RoboDK station: kr30 cnc template 7 axis 2.rdk

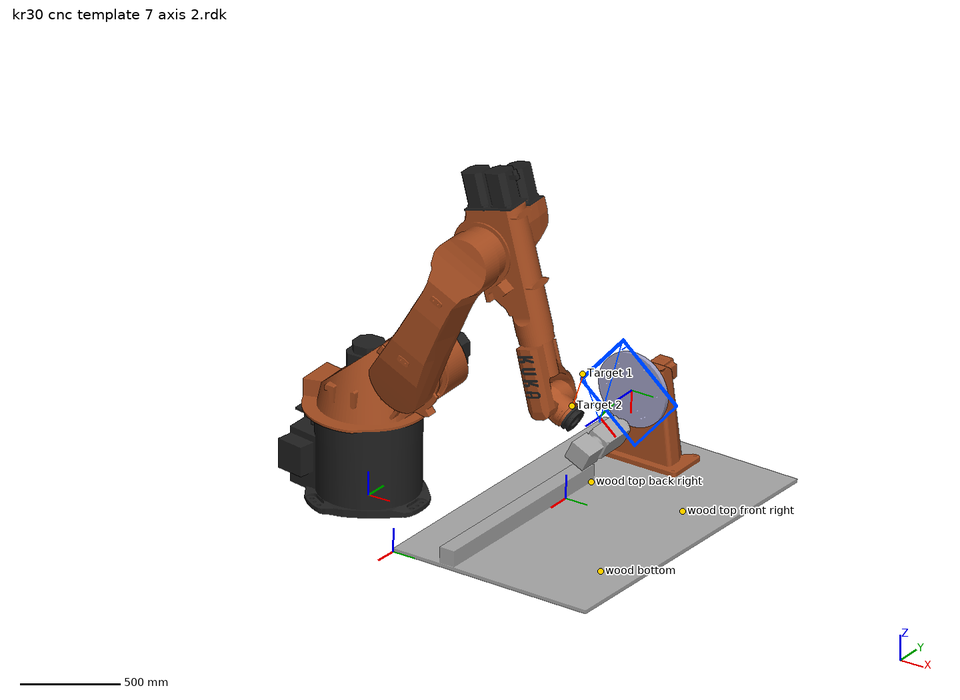
[picture v0: the station drawn from its stored meshes, robots at their saved joint values, targets as dots, program paths as lines]
Station kr30 cnc template 7 axis 2. Poses are relative to the parent item; angles as X-Y-Z fixed-axis rotations.
  - frame KUKA KR 30 HA Base at (0, 0, 0) mm
    - robot KUKA KR 30 HA: 6 axes, payload 30 kg, reach 2033 mm, repeatability 0.05 mm, weight 665 kg
        modified DH rows (alpha deg, a mm, theta deg, d mm): 0, 0, 0, 815; -90, 350, 0, 0; 0, 850, -90, 0; -90, 145, 0, 820; 90, 0, 0, 0; -90, 0, 180, 170
        joint limits [-185, -135, -120, -350, -119, -350] to [185, 35, 158, 350, 119, 350]; home [0, -90, 90, 0, 0, 0]; saved at [-1.685, -62.909, 138.513, -0.146, -48.713, -90.115]
      - tool rc90 spindle mm, TCP at (267.95, 0.68, 160.99) mm, rotated rx 0 ry 90 rz 0 deg, size 110 x 421.3 x 118 mm, geometry from rc90 spindle mm.stl
    - frame Tabletop at (921.82, -1104.91, 385) mm, rotated rx -0.93 ry -0.21 rz -89.9 deg
      - object tabletop CHECK HEIGHT at (-1839.9, 0, 0) mm, size 1839.9 x 1168.4 x 19 mm, geometry from kr30 tabletop mm.stl
      - object kr30 pipe jig base at (-1220, -610.6, 0) mm, size 1217.6 x 88.9 x 88.9 mm, geometry from kr30 pipe jig base.stl
      - frame Frame 3 at (-930, 400, 45) mm
      - target wood top back right (Cartesian target) at (-1141.49, 406.84, 52.26) mm, rotated rx 18.07 ry 89.88 rz 108.17 deg; joints [-2.086, -55.392, 143.759, 178.106, 87.553, -179.775] of KUKA KR 30 HA
      - target wood bottom (Cartesian target) at (-376.62, 995.52, 35.89) mm, rotated rx 18.07 ry 89.88 rz 108.17 deg; joints [24.587, -27.296, 76.752, 211.623, 53.064, -199.759] of KUKA KR 30 HA
      - target wood top front right (Cartesian target) at (-1142.68, 960.22, 52.55) mm, rotated rx 18.06 ry 89.88 rz 108.16 deg; joints [-1.42, -37.516, 98.016, 178.579, 59.693, -179.129] of KUKA KR 30 HA
  - machining project Machining Settings: C:/Users/Research Office/Desktop/paulina a5.apt | rotZ(0) | rotX(0)*rotY(0)
  - frame KUKA KP1 MD250 Base at (1360.87, 339.35, 824.43) mm, rotated rx -93.1 ry 88.62 rz 178.42 deg
    - robot KUKA KP1 MD250: 1 axes, payload 250 kg
        modified DH rows (alpha deg, a mm, theta deg, d mm): 0, 0, 0, 0
        joint limits [-360] to [360]; home [0]; saved at [-57.717]
    - frame Frame 5 at (179.73, -160.64, 39.79) mm, rotated rx 0 ry 0 rz 50 deg
      - target Target 1 (Cartesian target) at (-214.1, 84.73, -7.48) mm, rotated rx -180 ry 0 rz 150.96 deg; joints [-1.66, -91.883, 138.777, -0.061, 23.524, -90.098, -57.717] of KUKA KR 30 HA
      - target Target 2 (Cartesian target) at (-120.32, 1.96, 112.71) mm, rotated rx 180 ry 0 rz 142.66 deg; joints [4.871, -81.16, 137.42, -3.434, 22.572, -80.574, -143.17] of KUKA KR 30 HA
  - program Machining (635 instructions, listed below)
  - program sync move test (5 instructions, listed below)
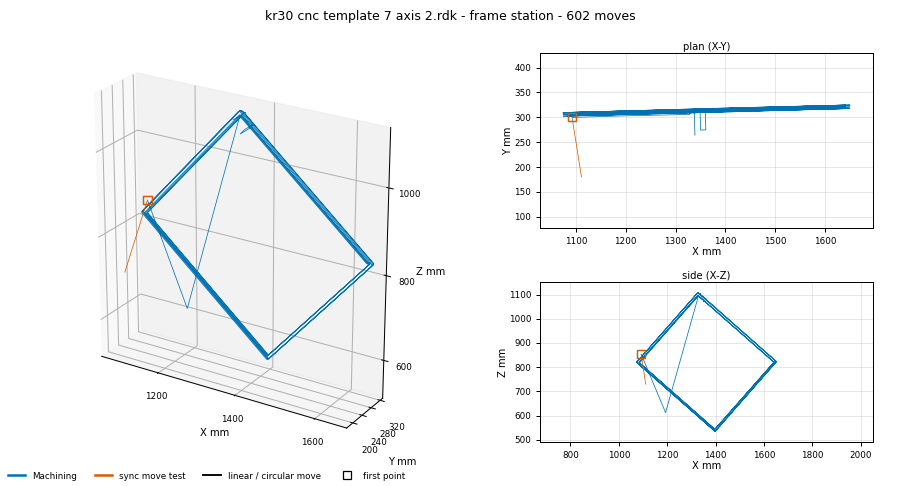
[picture p0: tool path of kr30 cnc template 7 axis 2.rdk in frame station, 602 of 602 moves have a stored position in this frame; points joined in program order, loops and branches not executed]

--- program Machining (robot KUKA KR 30 HA) ---
  Smooth(10)
  Print: /'1001'
  Print: /''
  Print: /'diagonal cut'
  Set speed (100.0 mm/s)
  Set Tool: rc90 spindle mm
  Set Ref.: Frame 5
  Show rc90 spindle mm
  MoveJ 1 to (-214.1, 84.73, -7.48) mm, rotated rx -180 ry 0 rz 150.96 deg; joints [-1.66, -91.883, 138.777, -0.061, 23.524, -90.098, -57.717]
  Set speed (38.1 mm/s)
  MoveL to (21.22, -29.86, -7.48) mm, rotated rx 180 ry 0 rz -151.32 deg; joints [-1.66, -91.883, 138.777, -0.061, 23.524, -90.098, -57.717]
  MoveL 1470 to (-195.61, 421.25, -7.47) mm, rotated rx 180 ry 0 rz 74.1 deg; joints [-1.66, -91.899, 138.812, -0.061, 23.524, -90.098, -57.737]
  Set speed (25.4 mm/s)
  MoveL 1471 to (-195.61, 421.25, -9.84) mm, rotated rx -180 ry 0 rz 74.1 deg; joints [-1.797, -91.898, 138.811, 0.054, 23.524, -90.333, -57.737]
  MoveL 1472 to (-195.61, 421.89, -10.47) mm, rotated rx 180 ry 0 rz 74.1 deg; joints [-1.834, -91.952, 138.836, 0.085, 23.524, -90.397, -57.707]
  Set speed (38.1 mm/s)
  MoveL 1473 to (-194.97, 422.52, -10.48) mm, rotated rx 180 ry 0 rz 74.1 deg; joints [-1.834, -91.991, 138.825, 0.086, 23.524, -90.397, -57.658]
  Set speed (76.2 mm/s)
  MoveL 1474 to (213.41, 422.52, -10.47) mm, rotated rx -180 ry 0 rz 74.1 deg; joints [-1.774, -87.647, 118.581, 0.214, 23.524, -90.444, -41.757]
  MoveL 1475 to (213.89, 422.53, -10.47) mm, rotated rx 180 ry 0 rz 74.1 deg; joints [-1.774, -87.649, 118.56, 0.214, 23.524, -90.445, -41.735]
  MoveL 1476 to (214.13, 422.55, -10.47) mm, rotated rx -180 ry 0 rz 74.1 deg; joints [-1.774, -87.652, 118.551, 0.214, 23.524, -90.445, -41.723]
  MoveL 1477 to (214.37, 422.59, -10.47) mm, rotated rx 180 ry 0 rz 74.1 deg; joints [-1.774, -87.656, 118.543, 0.214, 23.524, -90.445, -41.711]
  MoveL 1478 to (214.61, 422.65, -10.47) mm, rotated rx -180 ry 0 rz 74.1 deg; joints [-1.774, -87.662, 118.536, 0.215, 23.524, -90.445, -41.698]
  MoveL 1479 to (214.85, 422.74, -10.47) mm, rotated rx -180 ry 0 rz 74.1 deg; joints [-1.774, -87.67, 118.531, 0.215, 23.524, -90.445, -41.684]
  MoveL 1480 to (215.09, 422.84, -10.47) mm, rotated rx 180 ry 0 rz 74.1 deg; joints [-1.774, -87.68, 118.526, 0.215, 23.524, -90.445, -41.67]
  MoveL 1481 to (215.34, 422.97, -10.47) mm, rotated rx -180 ry 0 rz 74.1 deg; joints [-1.774, -87.691, 118.522, 0.215, 23.524, -90.445, -41.654]
  MoveL 1482 to (215.58, 423.13, -10.48) mm, rotated rx -180 ry 0 rz 74.1 deg; joints [-1.774, -87.706, 118.521, 0.215, 23.524, -90.445, -41.638]
  MoveL 1483 to (215.82, 423.33, -10.47) mm, rotated rx -180 ry 0 rz 74.1 deg; joints [-1.774, -87.723, 118.521, 0.215, 23.524, -90.446, -41.621]
  MoveL 1484 to (215.96, 423.46, -10.48) mm, rotated rx 180 ry 0 rz 74.1 deg; joints [-1.774, -87.735, 118.521, 0.216, 23.525, -90.446, -41.611]
  MoveL 1485 to (216.09, 423.6, -10.48) mm, rotated rx -180 ry 0 rz 74.1 deg; joints [-1.774, -87.745, 118.521, 0.216, 23.528, -90.446, -41.603]
  MoveL 1486 to (216.2, 423.73, -10.48) mm, rotated rx -180 ry 0 rz 74.1 deg; joints [-1.774, -87.756, 118.521, 0.216, 23.532, -90.446, -41.596]
  MoveL 1487 to (216.3, 423.87, -10.48) mm, rotated rx -180 ry 0 rz 74.1 deg; joints [-1.774, -87.766, 118.521, 0.216, 23.536, -90.446, -41.59]
  MoveL 1488 to (216.39, 424.01, -10.47) mm, rotated rx -180 ry 0 rz 74.1 deg; joints [-1.774, -87.776, 118.521, 0.216, 23.541, -90.446, -41.586]
  MoveL 1489 to (216.47, 424.15, -10.47) mm, rotated rx -180 ry 0 rz 74.1 deg; joints [-1.774, -87.786, 118.521, 0.216, 23.547, -90.446, -41.582]
  MoveL 1490 to (216.69, 424.27, -10.47) mm, rotated rx 180 ry 0 rz 74.1 deg; joints [-1.774, -87.797, 118.518, 0.216, 23.547, -90.446, -41.568]
  MoveL 1491 to (219.83, 424.27, -10.48) mm, rotated rx -180 ry 0 rz 74.1 deg; joints [-1.774, -87.806, 118.385, 0.217, 23.547, -90.447, -41.425]
  MoveL 1492 to (220.05, 424.15, -10.47) mm, rotated rx -180 ry 0 rz 74.1 deg; joints [-1.774, -87.797, 118.369, 0.217, 23.547, -90.447, -41.419]
  MoveL 1493 to (220.05, 53.41, -10.48) mm, rotated rx 180 ry 0 rz 74.1 deg; joints [-1.728, -59.035, 99.349, 0.059, 23.547, -90.273, -51.16]
  MoveL 1494 to (219.83, 53.18, -10.47) mm, rotated rx 180 ry 0 rz 74.1 deg; joints [-1.728, -59.018, 99.35, 0.059, 23.547, -90.272, -51.179]
  MoveL 1495 to (-199.12, 53.18, -10.48) mm, rotated rx 180 ry 0 rz 74.1 deg; joints [-1.791, -64.086, 127.611, -0.153, 23.547, -90.132, -74.372]
  MoveL 1496 to (-199.7, 53.17, -10.48) mm, rotated rx -180 ry 0 rz 74.1 deg; joints [-1.791, -64.101, 127.652, -0.153, 23.547, -90.132, -74.398]
  MoveL 1497 to (-199.9, 53.41, -10.48) mm, rotated rx -180 ry 0 rz 74.1 deg; joints [-1.791, -64.122, 127.672, -0.153, 23.545, -90.132, -74.394]
  MoveL 1498 to (-199.9, 424.15, -10.48) mm, rotated rx -180 ry 0 rz 74.1 deg; joints [-1.835, -92.249, 139.152, 0.086, 23.545, -90.399, -57.747]
  MoveL 1499 to (-199.7, 424.27, -10.48) mm, rotated rx 180 ry 0 rz 74.1 deg; joints [-1.835, -92.255, 139.146, 0.086, 23.545, -90.399, -57.735]
  MoveL 1500 to (-198.11, 424.27, -10.48) mm, rotated rx -180 ry 0 rz 74.1 deg; joints [-1.835, -92.216, 139.057, 0.086, 23.545, -90.399, -57.686]
  MoveL 1501 to (-197.87, 424.15, -10.47) mm, rotated rx -180 ry 0 rz 74.1 deg; joints [-1.835, -92.2, 139.04, 0.086, 23.545, -90.399, -57.685]
  MoveL 1502 to (-197.73, 423.93, -10.48) mm, rotated rx 180 ry 0 rz 74.1 deg; joints [-1.835, -92.178, 139.024, 0.086, 23.545, -90.399, -57.691]
  MoveL 1503 to (-197.57, 423.71, -10.48) mm, rotated rx -180 ry 0 rz 74.1 deg; joints [-1.835, -92.155, 139.006, 0.086, 23.545, -90.398, -57.696]
  MoveL 1504 to (-197.38, 423.49, -10.48) mm, rotated rx 180 ry 0 rz 74.1 deg; joints [-1.835, -92.131, 138.987, 0.086, 23.545, -90.398, -57.7]
  MoveL 1505 to (-197.14, 423.27, -10.47) mm, rotated rx -180 ry 0 rz 74.1 deg; joints [-1.834, -92.107, 138.966, 0.086, 23.545, -90.398, -57.703]
  MoveL 1506 to (-196.96, 423.13, -10.48) mm, rotated rx 180 ry 0 rz 74.1 deg; joints [-1.834, -92.09, 138.95, 0.086, 23.545, -90.398, -57.704]
  MoveL 1507 to (-196.78, 423, -10.47) mm, rotated rx -180 ry 0 rz 74.1 deg; joints [-1.834, -92.076, 138.935, 0.086, 23.545, -90.398, -57.704]
  MoveL 1508 to (-196.6, 422.9, -10.48) mm, rotated rx -180 ry 0 rz 74.1 deg; joints [-1.834, -92.062, 138.921, 0.086, 23.545, -90.398, -57.704]
  MoveL 1509 to (-196.42, 422.81, -10.48) mm, rotated rx -180 ry 0 rz 74.1 deg; joints [-1.834, -92.05, 138.908, 0.086, 23.545, -90.397, -57.702]
  MoveL 1510 to (-196.18, 422.71, -10.47) mm, rotated rx 180 ry 0 rz 74.1 deg; joints [-1.834, -92.036, 138.891, 0.086, 23.545, -90.397, -57.699]
  MoveL 1511 to (-195.93, 422.63, -10.48) mm, rotated rx 180 ry 0 rz 74.1 deg; joints [-1.834, -92.023, 138.874, 0.086, 23.545, -90.397, -57.696]
  MoveL 1512 to (-195.69, 422.58, -10.48) mm, rotated rx 180 ry 0 rz 74.1 deg; joints [-1.834, -92.013, 138.859, 0.086, 23.545, -90.397, -57.691]
  MoveL 1513 to (-195.45, 422.54, -10.48) mm, rotated rx 180 ry 0 rz 74.1 deg; joints [-1.834, -92.004, 138.844, 0.086, 23.545, -90.397, -57.685]
  MoveL 1514 to (-195.21, 422.52, -10.48) mm, rotated rx 180 ry 0 rz 74.1 deg; joints [-1.834, -91.996, 138.83, 0.086, 23.545, -90.397, -57.678]
  MoveL 1515 to (-194.97, 422.52, -10.48) mm, rotated rx -180 ry 0 rz 74.1 deg; joints [-1.834, -91.99, 138.817, 0.086, 23.545, -90.397, -57.671]
  Set speed (38.1 mm/s)
  MoveL 1516 to (-194.97, 421.25, -10.47) mm, rotated rx -180 ry 0 rz 74.1 deg; joints [-1.833, -91.882, 138.768, 0.085, 23.545, -90.396, -57.73]
  MoveL 1517 to (-195.61, 421.25, -10.48) mm, rotated rx -180 ry 0 rz 74.1 deg; joints [-1.834, -91.897, 138.803, 0.084, 23.545, -90.396, -57.75]
  Set speed (25.4 mm/s)
  MoveL 1518 to (-195.61, 421.25, -12.84) mm, rotated rx -180 ry 0 rz 74.1 deg; joints [-1.971, -91.896, 138.802, 0.199, 23.545, -90.631, -57.75]
  MoveL 1519 to (-195.61, 421.89, -13.47) mm, rotated rx -180 ry 0 rz 74.1 deg; joints [-2.008, -91.95, 138.826, 0.231, 23.545, -90.694, -57.72]
  Set speed (38.1 mm/s)
  MoveL 1520 to (-194.97, 422.52, -13.47) mm, rotated rx -180 ry 0 rz 74.1 deg; joints [-2.008, -91.989, 138.815, 0.232, 23.545, -90.695, -57.671]
  Set speed (76.2 mm/s)
  MoveL 1521 to (213.41, 422.52, -13.47) mm, rotated rx -180 ry 0 rz 74.1 deg; joints [-1.922, -87.638, 118.566, 0.429, 23.545, -90.761, -41.772]
  MoveL 1522 to (213.89, 422.53, -13.47) mm, rotated rx -180 ry 0 rz 74.1 deg; joints [-1.921, -87.64, 118.546, 0.429, 23.545, -90.762, -41.75]
  MoveL 1523 to (214.13, 422.55, -13.47) mm, rotated rx 180 ry 0 rz 74.1 deg; joints [-1.921, -87.642, 118.537, 0.429, 23.545, -90.762, -41.738]
  MoveL 1524 to (214.37, 422.59, -13.47) mm, rotated rx 180 ry 0 rz 74.1 deg; joints [-1.921, -87.647, 118.529, 0.429, 23.545, -90.762, -41.726]
  MoveL 1525 to (214.61, 422.65, -13.47) mm, rotated rx -180 ry 0 rz 74.1 deg; joints [-1.921, -87.653, 118.522, 0.429, 23.545, -90.762, -41.713]
  MoveL 1526 to (214.85, 422.74, -13.47) mm, rotated rx 180 ry 0 rz 74.1 deg; joints [-1.921, -87.66, 118.516, 0.43, 23.545, -90.762, -41.7]
  MoveL 1527 to (215.09, 422.84, -13.47) mm, rotated rx 180 ry 0 rz 74.1 deg; joints [-1.921, -87.67, 118.511, 0.43, 23.545, -90.762, -41.685]
  MoveL 1528 to (215.34, 422.97, -13.48) mm, rotated rx -180 ry 0 rz 74.1 deg; joints [-1.921, -87.682, 118.508, 0.43, 23.545, -90.763, -41.67]
  MoveL 1529 to (215.58, 423.13, -13.47) mm, rotated rx 180 ry 0 rz 74.1 deg; joints [-1.921, -87.696, 118.506, 0.43, 23.545, -90.763, -41.654]
  MoveL 1530 to (215.82, 423.33, -13.47) mm, rotated rx -180 ry 0 rz 74.1 deg; joints [-1.922, -87.714, 118.506, 0.431, 23.545, -90.763, -41.636]
  MoveL 1531 to (215.96, 423.46, -13.47) mm, rotated rx -180 ry 0 rz 74.1 deg; joints [-1.922, -87.725, 118.506, 0.431, 23.547, -90.763, -41.626]
  MoveL 1532 to (216.09, 423.6, -13.47) mm, rotated rx -180 ry 0 rz 74.1 deg; joints [-1.922, -87.736, 118.506, 0.431, 23.549, -90.763, -41.618]
  MoveL 1533 to (216.2, 423.73, -13.47) mm, rotated rx 180 ry 0 rz 74.1 deg; joints [-1.922, -87.747, 118.507, 0.431, 23.552, -90.763, -41.611]
  MoveL 1534 to (216.3, 423.87, -13.47) mm, rotated rx -180 ry 0 rz 74.1 deg; joints [-1.922, -87.757, 118.507, 0.431, 23.557, -90.763, -41.605]
  MoveL 1535 to (216.39, 424.01, -13.47) mm, rotated rx -180 ry 0 rz 74.1 deg; joints [-1.922, -87.767, 118.507, 0.431, 23.562, -90.763, -41.601]
  MoveL 1536 to (216.47, 424.15, -13.47) mm, rotated rx -180 ry 0 rz 74.1 deg; joints [-1.922, -87.776, 118.507, 0.431, 23.568, -90.763, -41.597]
  MoveL 1537 to (216.69, 424.27, -13.47) mm, rotated rx -180 ry 0 rz 74.1 deg; joints [-1.922, -87.787, 118.504, 0.432, 23.568, -90.764, -41.583]
  MoveL 1538 to (219.83, 424.27, -13.47) mm, rotated rx -180 ry 0 rz 74.1 deg; joints [-1.921, -87.797, 118.371, 0.433, 23.568, -90.765, -41.441]
  MoveL 1539 to (220.05, 424.15, -13.47) mm, rotated rx -180 ry 0 rz 74.1 deg; joints [-1.921, -87.788, 118.355, 0.433, 23.567, -90.765, -41.434]
  MoveL 1540 to (220.05, 53.41, -13.48) mm, rotated rx -180 ry 0 rz 74.1 deg; joints [-1.843, -59.027, 99.34, 0.185, 23.567, -90.49, -51.179]
  MoveL 1541 to (219.83, 53.18, -13.47) mm, rotated rx -180 ry 0 rz 74.1 deg; joints [-1.843, -59.01, 99.341, 0.185, 23.567, -90.49, -51.198]
  MoveL 1542 to (-197.29, 53.18, -13.48) mm, rotated rx -180 ry 0 rz 74.1 deg; joints [-1.931, -64.037, 127.476, -0.133, 23.567, -90.29, -74.307]
  MoveL 1543 to (-197.94, 53.18, -13.48) mm, rotated rx 180 ry 0 rz 74.1 deg; joints [-1.932, -64.054, 127.523, -0.134, 23.567, -90.29, -74.336]
  MoveL 1544 to (-198.16, 53.41, -13.48) mm, rotated rx -180 ry 0 rz 74.1 deg; joints [-1.932, -64.076, 127.544, -0.134, 23.567, -90.29, -74.335]
  MoveL 1545 to (-198.16, 424.15, -13.48) mm, rotated rx -180 ry 0 rz 74.1 deg; joints [-2.01, -92.205, 139.045, 0.232, 23.567, -90.697, -57.707]
  MoveL 1546 to (-198.01, 424.27, -13.48) mm, rotated rx -180 ry 0 rz 74.1 deg; joints [-2.01, -92.211, 139.042, 0.233, 23.567, -90.698, -57.697]
  MoveL 1547 to (-197.87, 424.15, -13.47) mm, rotated rx -180 ry 0 rz 74.1 deg; joints [-2.009, -92.198, 139.029, 0.233, 23.567, -90.697, -57.698]
  MoveL 1548 to (-197.73, 423.93, -13.47) mm, rotated rx -180 ry 0 rz 74.1 deg; joints [-2.009, -92.176, 139.013, 0.232, 23.567, -90.697, -57.705]
  MoveL 1549 to (-197.57, 423.71, -13.48) mm, rotated rx -180 ry 0 rz 74.1 deg; joints [-2.009, -92.153, 138.996, 0.232, 23.567, -90.697, -57.71]
  MoveL 1550 to (-197.38, 423.49, -13.48) mm, rotated rx -180 ry 0 rz 74.1 deg; joints [-2.009, -92.129, 138.977, 0.232, 23.567, -90.696, -57.714]
  MoveL 1551 to (-197.22, 423.33, -13.47) mm, rotated rx 180 ry 0 rz 74.1 deg; joints [-2.009, -92.112, 138.962, 0.232, 23.567, -90.696, -57.716]
  MoveL 1552 to (-197.14, 423.27, -13.48) mm, rotated rx -180 ry 0 rz 74.1 deg; joints [-2.009, -92.105, 138.955, 0.232, 23.567, -90.696, -57.717]
  MoveL 1553 to (-196.96, 423.13, -13.48) mm, rotated rx -180 ry 0 rz 74.1 deg; joints [-2.009, -92.088, 138.94, 0.232, 23.567, -90.696, -57.718]
  MoveL 1554 to (-196.78, 423, -13.47) mm, rotated rx -180 ry 0 rz 74.1 deg; joints [-2.009, -92.073, 138.925, 0.231, 23.567, -90.696, -57.718]
  MoveL 1555 to (-196.6, 422.9, -13.47) mm, rotated rx -180 ry 0 rz 74.1 deg; joints [-2.008, -92.06, 138.911, 0.231, 23.567, -90.695, -57.718]
  MoveL 1556 to (-196.42, 422.81, -13.47) mm, rotated rx 180 ry 0 rz 74.1 deg; joints [-2.008, -92.048, 138.897, 0.231, 23.567, -90.695, -57.716]
  MoveL 1557 to (-196.18, 422.71, -13.47) mm, rotated rx -180 ry 0 rz 74.1 deg; joints [-2.008, -92.034, 138.88, 0.231, 23.567, -90.695, -57.713]
  MoveL 1558 to (-195.93, 422.63, -13.47) mm, rotated rx 180 ry 0 rz 74.1 deg; joints [-2.008, -92.021, 138.864, 0.231, 23.567, -90.695, -57.709]
  MoveL 1559 to (-195.69, 422.58, -13.47) mm, rotated rx -180 ry 0 rz 74.1 deg; joints [-2.008, -92.011, 138.849, 0.231, 23.567, -90.695, -57.705]
  MoveL 1560 to (-195.45, 422.54, -13.48) mm, rotated rx 180 ry 0 rz 74.1 deg; joints [-2.008, -92.002, 138.834, 0.231, 23.567, -90.695, -57.699]
  MoveL 1561 to (-195.21, 422.52, -13.48) mm, rotated rx -180 ry 0 rz 74.1 deg; joints [-2.008, -91.994, 138.82, 0.231, 23.567, -90.695, -57.692]
  MoveL 1562 to (-194.97, 422.52, -13.47) mm, rotated rx 180 ry 0 rz 74.1 deg; joints [-2.008, -91.988, 138.806, 0.232, 23.567, -90.695, -57.685]
  Set speed (38.1 mm/s)
  MoveL 1563 to (-194.97, 421.25, -13.47) mm, rotated rx -180 ry 0 rz 74.1 deg; joints [-2.007, -91.88, 138.757, 0.23, 23.567, -90.693, -57.744]
  MoveL 1564 to (-195.61, 421.25, -13.47) mm, rotated rx 180 ry 0 rz 74.1 deg; joints [-2.008, -91.895, 138.792, 0.23, 23.567, -90.693, -57.764]
  Set speed (25.4 mm/s)
  MoveL 1565 to (-195.61, 421.25, -15.84) mm, rotated rx 180 ry 0 rz 74.1 deg; joints [-2.145, -91.894, 138.791, 0.344, 23.567, -90.927, -57.764]
  MoveL 1566 to (-195.61, 421.89, -16.48) mm, rotated rx 180 ry 0 rz 74.1 deg; joints [-2.182, -91.948, 138.815, 0.376, 23.567, -90.992, -57.734]
  Set speed (38.1 mm/s)
  MoveL 1567 to (-194.97, 422.52, -16.47) mm, rotated rx 180 ry 0 rz 74.1 deg; joints [-2.182, -91.986, 138.805, 0.378, 23.567, -90.993, -57.684]
  Set speed (76.2 mm/s)
  MoveL 1568 to (213.41, 422.52, -16.47) mm, rotated rx -180 ry 0 rz 74.1 deg; joints [-2.069, -87.627, 118.551, 0.643, 23.567, -91.078, -41.789]
  MoveL 1569 to (213.89, 422.53, -16.47) mm, rotated rx -180 ry 0 rz 74.1 deg; joints [-2.069, -87.629, 118.531, 0.643, 23.568, -91.078, -41.767]
  MoveL 1570 to (214.13, 422.55, -16.47) mm, rotated rx -180 ry 0 rz 74.1 deg; joints [-2.069, -87.632, 118.522, 0.643, 23.567, -91.078, -41.755]
  MoveL 1571 to (214.37, 422.59, -16.47) mm, rotated rx -180 ry 0 rz 74.1 deg; joints [-2.069, -87.636, 118.514, 0.643, 23.567, -91.078, -41.743]
  MoveL 1572 to (214.61, 422.65, -16.47) mm, rotated rx 180 ry 0 rz 74.1 deg; joints [-2.069, -87.642, 118.507, 0.644, 23.567, -91.078, -41.73]
  MoveL 1573 to (214.85, 422.74, -16.47) mm, rotated rx 180 ry 0 rz 74.1 deg; joints [-2.069, -87.65, 118.501, 0.644, 23.567, -91.079, -41.716]
  MoveL 1574 to (215.09, 422.84, -16.48) mm, rotated rx 180 ry 0 rz 74.1 deg; joints [-2.069, -87.66, 118.496, 0.644, 23.567, -91.079, -41.701]
  MoveL 1575 to (215.34, 422.97, -16.47) mm, rotated rx -180 ry 0 rz 74.1 deg; joints [-2.069, -87.672, 118.493, 0.645, 23.567, -91.079, -41.686]
  MoveL 1576 to (215.58, 423.13, -16.47) mm, rotated rx -180 ry 0 rz 74.1 deg; joints [-2.069, -87.686, 118.491, 0.645, 23.567, -91.08, -41.67]
  MoveL 1577 to (215.82, 423.33, -16.47) mm, rotated rx -180 ry 0 rz 74.1 deg; joints [-2.069, -87.703, 118.491, 0.646, 23.567, -91.08, -41.652]
  MoveL 1578 to (215.96, 423.46, -16.47) mm, rotated rx 180 ry 0 rz 74.1 deg; joints [-2.069, -87.715, 118.491, 0.646, 23.569, -91.08, -41.643]
  MoveL 1579 to (216.09, 423.6, -16.48) mm, rotated rx 180 ry 0 rz 74.1 deg; joints [-2.069, -87.726, 118.491, 0.646, 23.572, -91.08, -41.634]
  MoveL 1580 to (216.2, 423.73, -16.47) mm, rotated rx -180 ry 0 rz 74.1 deg; joints [-2.069, -87.736, 118.491, 0.646, 23.575, -91.08, -41.627]
  MoveL 1581 to (216.3, 423.87, -16.47) mm, rotated rx -180 ry 0 rz 74.1 deg; joints [-2.069, -87.746, 118.491, 0.646, 23.579, -91.08, -41.622]
  MoveL 1582 to (216.39, 424.01, -16.47) mm, rotated rx -180 ry 0 rz 74.1 deg; joints [-2.07, -87.756, 118.491, 0.646, 23.584, -91.08, -41.617]
  MoveL 1583 to (216.47, 424.15, -16.48) mm, rotated rx 180 ry 0 rz 74.1 deg; joints [-2.07, -87.766, 118.491, 0.646, 23.59, -91.08, -41.613]
  MoveL 1584 to (216.69, 424.27, -16.47) mm, rotated rx 180 ry 0 rz 74.1 deg; joints [-2.07, -87.777, 118.488, 0.646, 23.59, -91.081, -41.599]
  MoveL 1585 to (219.83, 424.27, -16.47) mm, rotated rx -180 ry 0 rz 74.1 deg; joints [-2.069, -87.787, 118.356, 0.649, 23.59, -91.082, -41.457]
  MoveL 1586 to (220.05, 424.15, -16.47) mm, rotated rx 180 ry 0 rz 74.1 deg; joints [-2.069, -87.777, 118.34, 0.649, 23.589, -91.082, -41.45]
  MoveL 1587 to (220.05, 53.41, -16.48) mm, rotated rx 180 ry 0 rz 74.1 deg; joints [-1.957, -59.019, 99.329, 0.31, 23.589, -90.707, -51.199]
  MoveL 1588 to (219.83, 53.17, -16.48) mm, rotated rx -180 ry 0 rz 74.1 deg; joints [-1.957, -59.001, 99.33, 0.309, 23.589, -90.707, -51.218]
  MoveL 1589 to (-196.42, 53.18, -16.48) mm, rotated rx 180 ry 0 rz 74.1 deg; joints [-2.072, -64.014, 127.409, -0.114, 23.589, -90.448, -74.285]
  MoveL 1590 to (-196.42, 53.41, -16.48) mm, rotated rx 180 ry 0 rz 74.1 deg; joints [-2.072, -64.03, 127.415, -0.114, 23.589, -90.448, -74.275]
  MoveL 1591 to (-196.42, 422.66, -16.48) mm, rotated rx -180 ry 0 rz 74.1 deg; joints [-2.183, -92.032, 138.881, 0.376, 23.589, -90.992, -57.737]
  MoveL 1592 to (-196.42, 422.81, -16.48) mm, rotated rx 180 ry 0 rz 74.1 deg; joints [-2.183, -92.045, 138.887, 0.377, 23.589, -90.993, -57.73]
  MoveL 1593 to (-196.18, 422.71, -16.48) mm, rotated rx 180 ry 0 rz 74.1 deg; joints [-2.182, -92.031, 138.87, 0.377, 23.589, -90.992, -57.727]
  MoveL 1594 to (-195.93, 422.63, -16.48) mm, rotated rx -180 ry 0 rz 74.1 deg; joints [-2.182, -92.018, 138.853, 0.377, 23.589, -90.992, -57.723]
  MoveL 1595 to (-195.69, 422.58, -16.47) mm, rotated rx -180 ry 0 rz 74.1 deg; joints [-2.182, -92.008, 138.838, 0.377, 23.589, -90.992, -57.718]
  MoveL 1596 to (-195.45, 422.54, -16.48) mm, rotated rx 180 ry 0 rz 74.1 deg; joints [-2.182, -91.999, 138.823, 0.377, 23.589, -90.992, -57.712]
  MoveL 1597 to (-195.21, 422.52, -16.48) mm, rotated rx -180 ry 0 rz 74.1 deg; joints [-2.182, -91.992, 138.809, 0.377, 23.589, -90.992, -57.706]
  MoveL 1598 to (-194.97, 422.52, -16.47) mm, rotated rx 180 ry 0 rz 74.1 deg; joints [-2.182, -91.986, 138.796, 0.377, 23.589, -90.992, -57.698]
  MoveL 1599 to (-164.9, 422.52, -17.53) mm, rotated rx 180 ry 0 rz 74.1 deg; joints [-2.229, -91.287, 137.144, 0.445, 23.589, -91.095, -56.745]
  MoveL 1600 to (213.41, 422.52, -17.52) mm, rotated rx -180 ry 0 rz 74.1 deg; joints [-2.121, -87.618, 118.537, 0.717, 23.589, -91.188, -41.805]
  MoveL 1601 to (213.89, 422.53, -17.52) mm, rotated rx 180 ry 0 rz 74.1 deg; joints [-2.121, -87.62, 118.516, 0.717, 23.589, -91.188, -41.783]
  MoveL 1602 to (214.13, 422.55, -17.52) mm, rotated rx -180 ry 0 rz 74.1 deg; joints [-2.121, -87.622, 118.507, 0.717, 23.589, -91.188, -41.771]
  MoveL 1603 to (214.37, 422.59, -17.52) mm, rotated rx -180 ry 0 rz 74.1 deg; joints [-2.121, -87.627, 118.499, 0.717, 23.589, -91.188, -41.759]
  MoveL 1604 to (214.61, 422.65, -17.52) mm, rotated rx 180 ry 0 rz 74.1 deg; joints [-2.121, -87.633, 118.492, 0.718, 23.589, -91.188, -41.746]
  MoveL 1605 to (214.85, 422.74, -17.52) mm, rotated rx -180 ry 0 rz 74.1 deg; joints [-2.121, -87.641, 118.486, 0.718, 23.589, -91.189, -41.732]
  MoveL 1606 to (215.09, 422.84, -17.52) mm, rotated rx 180 ry 0 rz 74.1 deg; joints [-2.121, -87.65, 118.482, 0.718, 23.589, -91.189, -41.718]
  MoveL 1607 to (215.34, 422.97, -17.52) mm, rotated rx -180 ry 0 rz 74.1 deg; joints [-2.121, -87.662, 118.478, 0.719, 23.589, -91.189, -41.703]
  MoveL 1608 to (215.58, 423.13, -17.52) mm, rotated rx -180 ry 0 rz 74.1 deg; joints [-2.121, -87.676, 118.476, 0.719, 23.589, -91.19, -41.686]
  MoveL 1609 to (215.82, 423.33, -17.52) mm, rotated rx -180 ry 0 rz 74.1 deg; joints [-2.121, -87.694, 118.476, 0.72, 23.589, -91.19, -41.669]
  MoveL 1610 to (215.96, 423.46, -17.52) mm, rotated rx -180 ry 0 rz 74.1 deg; joints [-2.121, -87.705, 118.476, 0.72, 23.591, -91.19, -41.659]
  MoveL 1611 to (216.09, 423.6, -17.52) mm, rotated rx 180 ry 0 rz 74.1 deg; joints [-2.121, -87.716, 118.476, 0.72, 23.594, -91.19, -41.651]
  MoveL 1612 to (216.2, 423.73, -17.52) mm, rotated rx 180 ry 0 rz 74.1 deg; joints [-2.121, -87.727, 118.477, 0.72, 23.597, -91.19, -41.644]
  MoveL 1613 to (216.3, 423.87, -17.52) mm, rotated rx 180 ry 0 rz 74.1 deg; joints [-2.121, -87.737, 118.477, 0.72, 23.601, -91.191, -41.638]
  MoveL 1614 to (216.39, 424.01, -17.52) mm, rotated rx -180 ry 0 rz 74.1 deg; joints [-2.121, -87.747, 118.477, 0.72, 23.606, -91.191, -41.633]
  MoveL 1615 to (216.47, 424.15, -17.52) mm, rotated rx -180 ry 0 rz 74.1 deg; joints [-2.121, -87.756, 118.477, 0.72, 23.612, -91.191, -41.629]
  MoveL 1616 to (216.69, 424.27, -17.52) mm, rotated rx 180 ry 0 rz 74.1 deg; joints [-2.121, -87.767, 118.474, 0.721, 23.612, -91.191, -41.615]
  MoveL 1617 to (219.83, 424.27, -17.52) mm, rotated rx 180 ry 0 rz 74.1 deg; joints [-2.121, -87.777, 118.341, 0.723, 23.612, -91.192, -41.473]
  MoveL 1618 to (220.05, 424.15, -17.52) mm, rotated rx 180 ry 0 rz 74.1 deg; joints [-2.121, -87.768, 118.326, 0.724, 23.612, -91.192, -41.466]
  MoveL 1619 to (220.05, 53.41, -17.52) mm, rotated rx -180 ry 0 rz 74.1 deg; joints [-1.996, -59.01, 99.319, 0.353, 23.612, -90.782, -51.22]
  MoveL 1620 to (219.83, 53.18, -17.52) mm, rotated rx 180 ry 0 rz 74.1 deg; joints [-1.996, -58.993, 99.321, 0.352, 23.612, -90.782, -51.239]
  MoveL 1621 to (-195.15, 53.18, -17.53) mm, rotated rx 180 ry 0 rz 74.1 deg; joints [-2.121, -63.98, 127.315, -0.107, 23.612, -90.504, -74.247]
  MoveL 1622 to (-195.65, 53.17, -17.52) mm, rotated rx 180 ry 0 rz 74.1 deg; joints [-2.121, -63.994, 127.351, -0.107, 23.612, -90.504, -74.269]
  MoveL 1623 to (-195.81, 53.41, -17.52) mm, rotated rx -180 ry 0 rz 74.1 deg; joints [-2.121, -64.014, 127.368, -0.107, 23.612, -90.504, -74.266]
  MoveL 1624 to (-195.81, 422.38, -17.53) mm, rotated rx -180 ry 0 rz 74.1 deg; joints [-2.243, -91.992, 138.827, 0.426, 23.612, -91.095, -57.745]
  MoveL 1625 to (-195.65, 422.57, -17.52) mm, rotated rx -180 ry 0 rz 74.1 deg; joints [-2.243, -92.004, 138.825, 0.427, 23.612, -91.095, -57.731]
  MoveL 1626 to (-195.48, 422.55, -17.52) mm, rotated rx -180 ry 0 rz 74.1 deg; joints [-2.243, -91.998, 138.815, 0.427, 23.612, -91.095, -57.727]
  MoveL 1627 to (-195.32, 422.53, -17.52) mm, rotated rx -180 ry 0 rz 74.1 deg; joints [-2.243, -91.993, 138.805, 0.427, 23.612, -91.095, -57.723]
  MoveL 1628 to (-195.15, 422.52, -17.53) mm, rotated rx 180 ry 0 rz 74.1 deg; joints [-2.243, -91.988, 138.796, 0.427, 23.612, -91.095, -57.718]
  MoveL 1629 to (-194.97, 422.52, -17.53) mm, rotated rx -180 ry 0 rz 74.1 deg; joints [-2.243, -91.984, 138.786, 0.427, 23.612, -91.095, -57.713]
  MoveL 1630 to (-164.9, 422.52, -17.52) mm, rotated rx 180 ry 0 rz 74.1 deg; joints [-2.229, -91.286, 137.134, 0.444, 23.612, -91.094, -56.759]
  Set speed (38.1 mm/s)
  MoveL 1631 to (-164.28, 421.77, -17.52) mm, rotated rx -180 ry 0 rz 74.1 deg; joints [-2.228, -91.208, 137.071, 0.443, 23.612, -91.093, -56.774]
  MoveL 1632 to (-164.81, 418.84, -17.52) mm, rotated rx 180 ry 0 rz 74.1 deg; joints [-2.226, -90.969, 136.984, 0.437, 23.612, -91.087, -56.926]
  MoveL 1633 to (-164.93, 418.21, -16.89) mm, rotated rx 180 ry 0 rz 74.1 deg; joints [-2.19, -90.919, 136.966, 0.405, 23.612, -91.023, -56.958]
  Set speed (100.0 mm/s)
  MoveL 1634 to (-164.93, 418.21, 24.52) mm, rotated rx -180 ry 0 rz 74.1 deg; joints [0.159, -90.892, 136.949, -1.635, 23.612, -86.951, -56.95]
  MoveL 1635 to (-164.87, 434.05, 24.53) mm, rotated rx -180 ry 0 rz 74.1 deg; joints [0.183, -92.247, 137.575, -1.706, 23.612, -86.872, -56.219]
  MoveL 1636 to (-164.87, 434.05, -6.52) mm, rotated rx -180 ry 0 rz 74.1 deg; joints [-1.602, -92.279, 137.596, -0.103, 23.612, -90.008, -56.229]
  Set speed (25.4 mm/s)
  MoveL 1637 to (-164.87, 434.05, -9.84) mm, rotated rx 180 ry 0 rz 74.1 deg; joints [-1.793, -92.278, 137.595, 0.069, 23.612, -90.343, -56.228]
  MoveL 1638 to (-164.72, 433.43, -10.47) mm, rotated rx -180 ry 0 rz 74.1 deg; joints [-1.83, -92.222, 137.562, 0.101, 23.612, -90.407, -56.252]
  Set speed (38.1 mm/s)
  MoveL 1639 to (-164.28, 431.48, -10.47) mm, rotated rx 180 ry 0 rz 74.1 deg; joints [-1.829, -92.044, 137.461, 0.1, 23.612, -90.405, -56.328]
  MoveL 1640 to (-164.9, 430.7, -10.47) mm, rotated rx 180 ry 0 rz 74.1 deg; joints [-1.829, -91.991, 137.463, 0.099, 23.612, -90.404, -56.384]
  Set speed (76.2 mm/s)
  MoveL 1641 to (-194.97, 430.7, -10.48) mm, rotated rx -180 ry 0 rz 74.1 deg; joints [-1.836, -92.69, 139.107, 0.092, 23.612, -90.404, -57.33]
  MoveL 1642 to (-202.2, 430.7, -10.48) mm, rotated rx 180 ry 0 rz 74.1 deg; joints [-1.837, -92.867, 139.506, 0.09, 23.612, -90.404, -57.551]
  MoveL 1643 to (-203.17, 430.7, -10.48) mm, rotated rx -180 ry 0 rz 74.1 deg; joints [-1.837, -92.89, 139.559, 0.09, 23.612, -90.404, -57.58]
  MoveL 1644 to (-203.41, 430.69, -10.47) mm, rotated rx 180 ry 0 rz 74.1 deg; joints [-1.838, -92.895, 139.571, 0.09, 23.612, -90.404, -57.589]
  MoveL 1645 to (-203.65, 430.65, -10.47) mm, rotated rx 180 ry 0 rz 74.1 deg; joints [-1.838, -92.898, 139.583, 0.09, 23.612, -90.404, -57.598]
  MoveL 1646 to (-203.89, 430.6, -10.48) mm, rotated rx -180 ry 0 rz 74.1 deg; joints [-1.838, -92.899, 139.595, 0.09, 23.612, -90.404, -57.607]
  MoveL 1647 to (-204.13, 430.52, -10.47) mm, rotated rx 180 ry 0 rz 74.1 deg; joints [-1.838, -92.899, 139.605, 0.089, 23.612, -90.404, -57.618]
  MoveL 1648 to (-204.42, 430.43, -10.48) mm, rotated rx 180 ry 0 rz 74.1 deg; joints [-1.838, -92.898, 139.618, 0.089, 23.612, -90.404, -57.632]
  MoveL 1649 to (-204.57, 430.37, -10.48) mm, rotated rx -180 ry 0 rz 74.1 deg; joints [-1.838, -92.897, 139.623, 0.089, 23.613, -90.404, -57.639]
  MoveL 1650 to (-204.72, 430.31, -10.48) mm, rotated rx -180 ry 0 rz 74.1 deg; joints [-1.838, -92.895, 139.629, 0.089, 23.612, -90.404, -57.646]
  MoveL 1651 to (-204.86, 430.23, -10.48) mm, rotated rx -180 ry 0 rz 74.1 deg; joints [-1.838, -92.892, 139.634, 0.089, 23.612, -90.404, -57.654]
  MoveL 1652 to (-205.01, 430.15, -10.48) mm, rotated rx -180 ry 0 rz 74.1 deg; joints [-1.838, -92.888, 139.639, 0.089, 23.612, -90.404, -57.663]
  MoveL 1653 to (-205.16, 430.05, -10.48) mm, rotated rx 180 ry 0 rz 74.1 deg; joints [-1.838, -92.884, 139.643, 0.089, 23.612, -90.404, -57.672]
  MoveL 1654 to (-205.3, 429.94, -10.48) mm, rotated rx 180 ry 0 rz 74.1 deg; joints [-1.838, -92.878, 139.647, 0.089, 23.612, -90.404, -57.681]
  MoveL 1655 to (-205.53, 429.75, -10.48) mm, rotated rx -180 ry 0 rz 74.1 deg; joints [-1.838, -92.867, 139.652, 0.088, 23.612, -90.404, -57.697]
  MoveL 1656 to (-205.75, 429.52, -10.48) mm, rotated rx -180 ry 0 rz 74.1 deg; joints [-1.838, -92.853, 139.656, 0.088, 23.612, -90.403, -57.715]
  MoveL 1657 to (-205.92, 429.3, -10.48) mm, rotated rx 180 ry 0 rz 74.1 deg; joints [-1.838, -92.838, 139.657, 0.088, 23.612, -90.403, -57.73]
  MoveL 1658 to (-206.06, 429.09, -10.48) mm, rotated rx -180 ry 0 rz 74.1 deg; joints [-1.838, -92.824, 139.656, 0.088, 23.612, -90.403, -57.745]
  MoveL 1659 to (-206.14, 428.95, -10.48) mm, rotated rx -180 ry 0 rz 74.1 deg; joints [-1.838, -92.814, 139.655, 0.088, 23.612, -90.403, -57.753]
  MoveL 1660 to (-206.21, 428.82, -10.47) mm, rotated rx 180 ry 0 rz 74.1 deg; joints [-1.838, -92.804, 139.654, 0.087, 23.612, -90.403, -57.762]
  MoveL 1661 to (-206.27, 428.69, -10.48) mm, rotated rx 180 ry 0 rz 74.1 deg; joints [-1.838, -92.794, 139.652, 0.087, 23.612, -90.403, -57.77]
  MoveL 1662 to (-206.32, 428.55, -10.48) mm, rotated rx -180 ry 0 rz 74.1 deg; joints [-1.838, -92.784, 139.65, 0.087, 23.612, -90.402, -57.778]
  MoveL 1663 to (-206.37, 428.42, -10.47) mm, rotated rx -180 ry 0 rz 74.1 deg; joints [-1.838, -92.773, 139.647, 0.087, 23.612, -90.402, -57.786]
  MoveL 1664 to (-206.41, 428.28, -10.48) mm, rotated rx -180 ry 0 rz 74.1 deg; joints [-1.838, -92.763, 139.644, 0.087, 23.612, -90.402, -57.793]
  MoveL 1665 to (-206.47, 428.01, -10.48) mm, rotated rx -180 ry 0 rz 74.1 deg; joints [-1.838, -92.741, 139.637, 0.087, 23.612, -90.402, -57.808]
  MoveL 1666 to (-206.5, 427.77, -10.48) mm, rotated rx -180 ry 0 rz 74.1 deg; joints [-1.838, -92.721, 139.63, 0.087, 23.612, -90.402, -57.82]
  MoveL 1667 to (-206.52, 427.53, -10.48) mm, rotated rx 180 ry 0 rz 74.1 deg; joints [-1.837, -92.701, 139.621, 0.086, 23.612, -90.401, -57.832]
  MoveL 1668 to (-206.52, 427.04, -10.47) mm, rotated rx 180 ry 0 rz 74.1 deg; joints [-1.837, -92.659, 139.603, 0.086, 23.612, -90.401, -57.855]
  MoveL 1669 to (-206.52, 50.21, -10.48) mm, rotated rx -180 ry 0 rz 74.1 deg; joints [-1.792, -64.093, 128.064, -0.158, 23.612, -90.128, -74.883]
  MoveL 1670 to (-206.51, 49.73, -10.48) mm, rotated rx 180 ry 0 rz 74.1 deg; joints [-1.792, -64.06, 128.052, -0.158, 23.612, -90.128, -74.904]
  MoveL 1671 to (-206.48, 49.48, -10.48) mm, rotated rx 180 ry 0 rz 74.1 deg; joints [-1.792, -64.042, 128.044, -0.159, 23.612, -90.128, -74.913]
  MoveL 1672 to (-206.43, 49.24, -10.48) mm, rotated rx 180 ry 0 rz 74.1 deg; joints [-1.792, -64.025, 128.035, -0.159, 23.612, -90.127, -74.922]
  MoveL 1673 to (-206.37, 49.02, -10.48) mm, rotated rx -180 ry 0 rz 74.1 deg; joints [-1.792, -64.008, 128.025, -0.159, 23.612, -90.127, -74.929]
  MoveL 1674 to (-206.28, 48.8, -10.48) mm, rotated rx -180 ry 0 rz 74.1 deg; joints [-1.792, -63.99, 128.014, -0.159, 23.612, -90.127, -74.936]
  MoveL 1675 to (-206.18, 48.57, -10.48) mm, rotated rx -180 ry 0 rz 74.1 deg; joints [-1.792, -63.972, 128.002, -0.159, 23.612, -90.127, -74.942]
  MoveL 1676 to (-206.06, 48.35, -10.48) mm, rotated rx -180 ry 0 rz 74.1 deg; joints [-1.792, -63.954, 127.988, -0.159, 23.612, -90.127, -74.946]
  MoveL 1677 to (-205.98, 48.22, -10.48) mm, rotated rx 180 ry 0 rz 74.1 deg; joints [-1.792, -63.943, 127.979, -0.159, 23.612, -90.127, -74.948]
  MoveL 1678 to (-205.88, 48.09, -10.48) mm, rotated rx -180 ry 0 rz 74.1 deg; joints [-1.792, -63.931, 127.969, -0.159, 23.612, -90.127, -74.95]
  MoveL 1679 to (-205.78, 47.96, -10.48) mm, rotated rx -180 ry 0 rz 74.1 deg; joints [-1.792, -63.92, 127.959, -0.159, 23.612, -90.127, -74.952]
  MoveL 1680 to (-205.66, 47.83, -10.48) mm, rotated rx -180 ry 0 rz 74.1 deg; joints [-1.792, -63.907, 127.948, -0.159, 23.612, -90.127, -74.952]
  MoveL 1681 to (-205.51, 47.67, -10.48) mm, rotated rx -180 ry 0 rz 74.1 deg; joints [-1.792, -63.892, 127.933, -0.159, 23.612, -90.127, -74.952]
  MoveL 1682 to (-205.35, 47.54, -10.48) mm, rotated rx -180 ry 0 rz 74.1 deg; joints [-1.792, -63.879, 127.918, -0.159, 23.612, -90.127, -74.952]
  MoveL 1683 to (-205.19, 47.42, -10.48) mm, rotated rx -180 ry 0 rz 74.1 deg; joints [-1.792, -63.866, 127.904, -0.159, 23.612, -90.127, -74.95]
  MoveL 1684 to (-205.03, 47.31, -10.48) mm, rotated rx 180 ry 0 rz 74.1 deg; joints [-1.792, -63.854, 127.89, -0.159, 23.612, -90.127, -74.948]
  MoveL 1685 to (-204.81, 47.18, -10.48) mm, rotated rx 180 ry 0 rz 74.1 deg; joints [-1.792, -63.839, 127.871, -0.159, 23.611, -90.127, -74.943]
  MoveL 1686 to (-204.58, 47.08, -10.48) mm, rotated rx -180 ry 0 rz 74.1 deg; joints [-1.792, -63.826, 127.853, -0.159, 23.611, -90.127, -74.938]
  MoveL 1687 to (-204.36, 46.99, -10.48) mm, rotated rx -180 ry 0 rz 74.1 deg; joints [-1.792, -63.814, 127.835, -0.159, 23.611, -90.127, -74.932]
  MoveL 1688 to (-204.13, 46.92, -10.48) mm, rotated rx -180 ry 0 rz 74.1 deg; joints [-1.791, -63.802, 127.818, -0.159, 23.603, -90.127, -74.918]
  MoveL 1689 to (-203.89, 46.87, -10.48) mm, rotated rx 180 ry 0 rz 74.1 deg; joints [-1.791, -63.792, 127.799, -0.159, 23.603, -90.127, -74.91]
  MoveL 1690 to (-203.65, 46.84, -10.48) mm, rotated rx -180 ry 0 rz 74.1 deg; joints [-1.791, -63.783, 127.781, -0.159, 23.603, -90.127, -74.901]
  MoveL 1691 to (-203.41, 46.83, -10.48) mm, rotated rx -180 ry 0 rz 74.1 deg; joints [-1.791, -63.776, 127.763, -0.158, 23.603, -90.127, -74.891]
  MoveL 1692 to (-203.17, 46.83, -10.48) mm, rotated rx 180 ry 0 rz 74.1 deg; joints [-1.791, -63.769, 127.746, -0.158, 23.603, -90.127, -74.88]
  MoveL 1693 to (222.09, 46.83, -10.47) mm, rotated rx 180 ry 0 rz 74.1 deg; joints [-1.728, -58.551, 98.86, 0.058, 23.603, -90.271, -51.212]
  MoveL 1694 to (223.29, 46.83, -10.47) mm, rotated rx -180 ry 0 rz 74.1 deg; joints [-1.728, -58.556, 98.788, 0.059, 23.603, -90.271, -51.135]
  MoveL 1695 to (223.53, 46.84, -10.48) mm, rotated rx -180 ry 0 rz 74.1 deg; joints [-1.728, -58.558, 98.774, 0.059, 23.603, -90.271, -51.12]
  MoveL 1696 to (223.77, 46.87, -10.48) mm, rotated rx -180 ry 0 rz 74.1 deg; joints [-1.728, -58.561, 98.761, 0.059, 23.604, -90.271, -51.105]
  MoveL 1697 to (224.01, 46.92, -10.47) mm, rotated rx -180 ry 0 rz 74.1 deg; joints [-1.728, -58.565, 98.75, 0.059, 23.604, -90.271, -51.088]
  MoveL 1698 to (224.24, 46.99, -10.48) mm, rotated rx -180 ry 0 rz 74.1 deg; joints [-1.728, -58.571, 98.74, 0.059, 23.604, -90.272, -51.073]
  MoveL 1699 to (224.46, 47.08, -10.47) mm, rotated rx -180 ry 0 rz 74.1 deg; joints [-1.728, -58.578, 98.731, 0.059, 23.604, -90.272, -51.057]
  MoveL 1700 to (224.69, 47.18, -10.48) mm, rotated rx 180 ry 0 rz 74.1 deg; joints [-1.728, -58.587, 98.723, 0.059, 23.604, -90.272, -51.04]
  MoveL 1701 to (224.92, 47.31, -10.47) mm, rotated rx -180 ry 0 rz 74.1 deg; joints [-1.728, -58.597, 98.717, 0.06, 23.604, -90.272, -51.024]
  MoveL 1702 to (225.07, 47.42, -10.48) mm, rotated rx -180 ry 0 rz 74.1 deg; joints [-1.728, -58.605, 98.713, 0.06, 23.604, -90.272, -51.012]
  MoveL 1703 to (225.23, 47.54, -10.48) mm, rotated rx -180 ry 0 rz 74.1 deg; joints [-1.728, -58.614, 98.71, 0.06, 23.604, -90.272, -51]
  MoveL 1704 to (225.39, 47.67, -10.47) mm, rotated rx 180 ry 0 rz 74.1 deg; joints [-1.728, -58.625, 98.708, 0.06, 23.604, -90.272, -50.986]
  MoveL 1705 to (225.55, 47.83, -10.47) mm, rotated rx 180 ry 0 rz 74.1 deg; joints [-1.727, -58.637, 98.707, 0.06, 23.604, -90.272, -50.974]
  MoveL 1706 to (225.66, 47.96, -10.47) mm, rotated rx 180 ry 0 rz 74.1 deg; joints [-1.727, -58.647, 98.707, 0.06, 23.604, -90.272, -50.964]
  MoveL 1707 to (225.77, 48.09, -10.47) mm, rotated rx -180 ry 0 rz 74.1 deg; joints [-1.727, -58.656, 98.707, 0.06, 23.604, -90.272, -50.955]
  MoveL 1708 to (225.86, 48.22, -10.47) mm, rotated rx 180 ry 0 rz 74.1 deg; joints [-1.727, -58.666, 98.709, 0.06, 23.604, -90.272, -50.947]
  MoveL 1709 to (225.94, 48.35, -10.47) mm, rotated rx -180 ry 0 rz 74.1 deg; joints [-1.727, -58.676, 98.711, 0.06, 23.604, -90.273, -50.939]
  MoveL 1710 to (226.07, 48.57, -10.48) mm, rotated rx 180 ry 0 rz 74.1 deg; joints [-1.727, -58.692, 98.715, 0.06, 23.605, -90.273, -50.928]
  MoveL 1711 to (226.17, 48.8, -10.47) mm, rotated rx 180 ry 0 rz 74.1 deg; joints [-1.727, -58.708, 98.721, 0.061, 23.605, -90.273, -50.917]
  MoveL 1712 to (226.25, 49.02, -10.48) mm, rotated rx 180 ry 0 rz 74.1 deg; joints [-1.728, -58.724, 98.728, 0.061, 23.605, -90.273, -50.908]
  MoveL 1713 to (226.31, 49.24, -10.48) mm, rotated rx 180 ry 0 rz 74.1 deg; joints [-1.728, -58.741, 98.736, 0.061, 23.605, -90.273, -50.9]
  MoveL 1714 to (226.36, 49.48, -10.48) mm, rotated rx 180 ry 0 rz 74.1 deg; joints [-1.728, -58.758, 98.745, 0.061, 23.606, -90.273, -50.893]
  MoveL 1715 to (226.39, 49.73, -10.47) mm, rotated rx -180 ry 0 rz 74.1 deg; joints [-1.728, -58.775, 98.756, 0.061, 23.606, -90.273, -50.886]
  MoveL 1716 to (226.4, 50.21, -10.48) mm, rotated rx 180 ry 0 rz 74.1 deg; joints [-1.728, -58.81, 98.781, 0.061, 23.606, -90.273, -50.877]
  MoveL 1717 to (226.4, 427.53, -10.47) mm, rotated rx 180 ry 0 rz 74.1 deg; joints [-1.73, -73.761, 98.781, -0.032, 51.624, -90.2, -63.944]
  MoveL 1718 to (226.39, 427.77, -10.47) mm, rotated rx -180 ry 0 rz 74.1 deg; joints [-1.73, -73.772, 98.781, -0.032, 51.636, -90.2, -63.944]
  MoveL 1719 to (226.37, 428.01, -10.48) mm, rotated rx -180 ry 0 rz 74.1 deg; joints [-1.73, -73.783, 98.781, -0.032, 51.649, -90.2, -63.947]
  MoveL 1720 to (226.34, 428.16, -10.47) mm, rotated rx -180 ry 0 rz 74.1 deg; joints [-1.73, -73.789, 98.781, -0.032, 51.658, -90.2, -63.95]
  MoveL 1721 to (226.31, 428.3, -10.47) mm, rotated rx 180 ry 0 rz 74.1 deg; joints [-1.73, -73.795, 98.781, -0.032, 51.668, -90.2, -63.953]
  MoveL 1722 to (226.27, 428.45, -10.47) mm, rotated rx -180 ry 0 rz 74.1 deg; joints [-1.73, -73.801, 98.781, -0.032, 51.678, -90.2, -63.958]
  MoveL 1723 to (226.22, 428.59, -10.47) mm, rotated rx -180 ry 0 rz 74.1 deg; joints [-1.73, -73.807, 98.781, -0.032, 51.689, -90.2, -63.963]
  MoveL 1724 to (226.16, 428.74, -10.47) mm, rotated rx -180 ry 0 rz 74.1 deg; joints [-1.73, -73.812, 98.781, -0.032, 51.7, -90.2, -63.969]
  MoveL 1725 to (226.1, 428.89, -10.47) mm, rotated rx 180 ry 0 rz 74.1 deg; joints [-1.73, -73.817, 98.781, -0.032, 51.713, -90.2, -63.976]
  MoveL 1726 to (226.03, 429.03, -10.48) mm, rotated rx 180 ry 0 rz 74.1 deg; joints [-1.73, -73.822, 98.781, -0.032, 51.726, -90.2, -63.984]
  MoveL 1727 to (225.94, 429.18, -10.48) mm, rotated rx 180 ry 0 rz 74.1 deg; joints [-1.73, -73.827, 98.781, -0.032, 51.739, -90.2, -63.994]
  MoveL 1728 to (225.82, 429.37, -10.47) mm, rotated rx -180 ry 0 rz 74.1 deg; joints [-1.73, -73.832, 98.781, -0.032, 51.759, -90.2, -64.008]
  MoveL 1729 to (225.67, 429.56, -10.47) mm, rotated rx 180 ry 0 rz 74.1 deg; joints [-1.73, -73.837, 98.781, -0.032, 51.78, -90.199, -64.024]
  MoveL 1730 to (225.5, 429.75, -10.48) mm, rotated rx -180 ry 0 rz 74.1 deg; joints [-1.73, -73.841, 98.781, -0.032, 51.804, -90.199, -64.044]
  MoveL 1731 to (225.29, 429.94, -10.47) mm, rotated rx -180 ry 0 rz 74.1 deg; joints [-1.73, -73.845, 98.781, -0.032, 51.83, -90.199, -64.067]
  MoveL 1732 to (225.13, 430.07, -10.47) mm, rotated rx -180 ry 0 rz 74.1 deg; joints [-1.73, -73.846, 98.781, -0.032, 51.85, -90.199, -64.085]
  MoveL 1733 to (224.97, 430.18, -10.47) mm, rotated rx -180 ry 0 rz 74.1 deg; joints [-1.73, -73.847, 98.781, -0.032, 51.868, -90.199, -64.102]
  MoveL 1734 to (224.81, 430.28, -10.47) mm, rotated rx -180 ry 0 rz 74.1 deg; joints [-1.73, -73.847, 98.781, -0.032, 51.886, -90.199, -64.12]
  MoveL 1735 to (224.65, 430.37, -10.48) mm, rotated rx 180 ry 0 rz 74.1 deg; joints [-1.73, -73.847, 98.782, -0.033, 51.903, -90.199, -64.138]
  MoveL 1736 to (224.49, 430.44, -10.48) mm, rotated rx -180 ry 0 rz 74.1 deg; joints [-1.73, -73.847, 98.783, -0.033, 51.918, -90.199, -64.154]
  MoveL 1737 to (224.33, 430.51, -10.48) mm, rotated rx 180 ry 0 rz 74.1 deg; joints [-1.73, -73.847, 98.785, -0.033, 51.932, -90.199, -64.17]
  MoveL 1738 to (224.17, 430.56, -10.47) mm, rotated rx -180 ry 0 rz 74.1 deg; joints [-1.73, -73.847, 98.788, -0.033, 51.944, -90.199, -64.185]
  MoveL 1739 to (224.01, 430.6, -10.47) mm, rotated rx -180 ry 0 rz 74.1 deg; joints [-1.73, -73.847, 98.791, -0.033, 51.956, -90.199, -64.199]
  MoveL 1740 to (223.77, 430.66, -10.47) mm, rotated rx 180 ry 0 rz 74.1 deg; joints [-1.73, -73.847, 98.797, -0.033, 51.971, -90.199, -64.22]
  MoveL 1741 to (223.53, 430.69, -10.48) mm, rotated rx 180 ry 0 rz 74.1 deg; joints [-1.73, -73.847, 98.803, -0.033, 51.983, -90.199, -64.239]
  MoveL 1742 to (223.29, 430.7, -10.47) mm, rotated rx -180 ry 0 rz 74.1 deg; joints [-1.73, -73.847, 98.811, -0.033, 51.993, -90.199, -64.258]
  MoveL 1743 to (223.05, 430.7, -10.47) mm, rotated rx -180 ry 0 rz 74.1 deg; joints [-1.73, -73.847, 98.82, -0.033, 52.002, -90.199, -64.275]
  MoveL 1744 to (-164.9, 430.7, -10.47) mm, rotated rx -180 ry 0 rz 74.1 deg; joints [-1.784, -86.616, 123.581, -0.089, 52.002, -90.208, -76.266]
  Set speed (38.1 mm/s)
  MoveL 1745 to (-165.25, 431.87, -10.47) mm, rotated rx 180 ry 0 rz 74.1 deg; joints [-1.784, -86.716, 123.626, -0.089, 52.002, -90.208, -76.212]
  MoveL 1746 to (-164.27, 432.52, -10.47) mm, rotated rx -180 ry 0 rz 74.1 deg; joints [-1.784, -86.718, 123.574, -0.088, 52.002, -90.209, -76.158]
  Set speed (25.4 mm/s)
  MoveL 1747 to (-164.27, 432.52, -12.84) mm, rotated rx -180 ry 0 rz 74.1 deg; joints [-1.902, -86.718, 123.573, -0.085, 52.002, -90.329, -76.158]
  MoveL 1748 to (-164.27, 431.89, -13.47) mm, rotated rx -180 ry 0 rz 74.1 deg; joints [-1.934, -86.672, 123.561, -0.085, 52.002, -90.361, -76.191]
  Set speed (38.1 mm/s)
  MoveL 1749 to (-164.9, 431.25, -13.48) mm, rotated rx -180 ry 0 rz 74.1 deg; joints [-1.934, -86.654, 123.589, -0.085, 52.003, -90.361, -76.238]
  Set speed (76.2 mm/s)
  MoveL 1750 to (-194.97, 431.25, -13.48) mm, rotated rx -180 ry 0 rz 74.1 deg; joints [-1.943, -88.044, 125.539, -0.09, 52.003, -90.366, -76.798]
  MoveL 1751 to (-201.24, 431.25, -13.47) mm, rotated rx -180 ry 0 rz 74.1 deg; joints [-1.945, -88.341, 125.946, -0.091, 52.003, -90.368, -76.908]
  MoveL 1752 to (-201.48, 431.25, -13.47) mm, rotated rx -180 ry 0 rz 74.1 deg; joints [-1.946, -88.352, 125.961, -0.091, 52.003, -90.368, -76.912]
  MoveL 1753 to (-201.72, 431.23, -13.47) mm, rotated rx -180 ry 0 rz 74.1 deg; joints [-1.946, -88.362, 125.977, -0.091, 52.003, -90.368, -76.918]
  MoveL 1754 to (-201.96, 431.19, -13.47) mm, rotated rx -180 ry 0 rz 74.1 deg; joints [-1.946, -88.371, 125.991, -0.091, 52.003, -90.368, -76.924]
  MoveL 1755 to (-202.2, 431.13, -13.48) mm, rotated rx 180 ry 0 rz 74.1 deg; joints [-1.946, -88.378, 126.006, -0.091, 52.003, -90.368, -76.931]
  MoveL 1756 to (-204.13, 430.52, -13.48) mm, rotated rx -180 ry 0 rz 74.1 deg; joints [-1.946, -88.426, 126.12, -0.092, 52.003, -90.368, -76.997]
  MoveL 1757 to (-204.42, 430.43, -13.48) mm, rotated rx 180 ry 0 rz 74.1 deg; joints [-1.946, -88.433, 126.137, -0.092, 52.003, -90.368, -77.007]
  MoveL 1758 to (-204.57, 430.37, -13.47) mm, rotated rx 180 ry 0 rz 74.1 deg; joints [-1.946, -88.436, 126.146, -0.092, 52.003, -90.368, -77.013]
  MoveL 1759 to (-204.72, 430.31, -13.47) mm, rotated rx 180 ry 0 rz 74.1 deg; joints [-1.946, -88.439, 126.154, -0.092, 52.003, -90.368, -77.019]
  MoveL 1760 to (-204.86, 430.23, -13.48) mm, rotated rx 180 ry 0 rz 74.1 deg; joints [-1.946, -88.44, 126.162, -0.092, 52.003, -90.368, -77.025]
  MoveL 1761 to (-205.01, 430.15, -13.47) mm, rotated rx 180 ry 0 rz 74.1 deg; joints [-1.946, -88.441, 126.17, -0.092, 52.003, -90.368, -77.032]
  MoveL 1762 to (-205.16, 430.05, -13.47) mm, rotated rx -180 ry 0 rz 74.1 deg; joints [-1.946, -88.441, 126.178, -0.093, 52.003, -90.368, -77.04]
  MoveL 1763 to (-205.3, 429.94, -13.47) mm, rotated rx -180 ry 0 rz 74.1 deg; joints [-1.947, -88.44, 126.185, -0.093, 52.003, -90.368, -77.048]
  MoveL 1764 to (-205.53, 429.75, -13.47) mm, rotated rx 180 ry 0 rz 74.1 deg; joints [-1.947, -88.437, 126.196, -0.093, 52.003, -90.368, -77.062]
  MoveL 1765 to (-205.75, 429.52, -13.47) mm, rotated rx -180 ry 0 rz 74.1 deg; joints [-1.947, -88.431, 126.207, -0.093, 52.003, -90.368, -77.079]
  MoveL 1766 to (-205.92, 429.3, -13.48) mm, rotated rx -180 ry 0 rz 74.1 deg; joints [-1.947, -88.424, 126.214, -0.093, 52.003, -90.367, -77.093]
  MoveL 1767 to (-206.06, 429.09, -13.47) mm, rotated rx 180 ry 0 rz 74.1 deg; joints [-1.947, -88.416, 126.219, -0.093, 52.003, -90.367, -77.107]
  MoveL 1768 to (-206.14, 428.95, -13.47) mm, rotated rx -180 ry 0 rz 74.1 deg; joints [-1.947, -88.41, 126.222, -0.093, 52.003, -90.367, -77.115]
  MoveL 1769 to (-206.21, 428.82, -13.47) mm, rotated rx -180 ry 0 rz 74.1 deg; joints [-1.947, -88.403, 126.224, -0.093, 52.003, -90.367, -77.124]
  MoveL 1770 to (-206.27, 428.69, -13.48) mm, rotated rx -180 ry 0 rz 74.1 deg; joints [-1.947, -88.397, 126.225, -0.093, 52.003, -90.367, -77.132]
  MoveL 1771 to (-206.32, 428.55, -13.48) mm, rotated rx 180 ry 0 rz 74.1 deg; joints [-1.947, -88.389, 126.226, -0.093, 52.003, -90.367, -77.14]
  MoveL 1772 to (-206.37, 428.42, -13.47) mm, rotated rx -180 ry 0 rz 74.1 deg; joints [-1.947, -88.382, 126.227, -0.094, 52.003, -90.367, -77.148]
  MoveL 1773 to (-206.41, 428.28, -13.47) mm, rotated rx 180 ry 0 rz 74.1 deg; joints [-1.947, -88.374, 126.227, -0.094, 52.003, -90.367, -77.156]
  MoveL 1774 to (-206.47, 428.01, -13.47) mm, rotated rx 180 ry 0 rz 74.1 deg; joints [-1.946, -88.358, 126.226, -0.094, 52.003, -90.367, -77.172]
  MoveL 1775 to (-206.5, 427.77, -13.47) mm, rotated rx -180 ry 0 rz 74.1 deg; joints [-1.946, -88.342, 126.224, -0.094, 52.003, -90.367, -77.185]
  MoveL 1776 to (-206.52, 427.53, -13.47) mm, rotated rx -180 ry 0 rz 74.1 deg; joints [-1.946, -88.326, 126.221, -0.094, 52.003, -90.367, -77.198]
  MoveL 1777 to (-206.52, 427.04, -13.47) mm, rotated rx -180 ry 0 rz 74.1 deg; joints [-1.946, -88.291, 126.212, -0.094, 52.003, -90.366, -77.224]
  MoveL 1778 to (-206.52, 50.21, -13.48) mm, rotated rx -180 ry 0 rz 74.1 deg; joints [-1.916, -65.223, 123.892, -0.265, 52.003, -90.179, -97.973]
  MoveL 1779 to (-206.51, 49.73, -13.47) mm, rotated rx -180 ry 0 rz 74.1 deg; joints [-1.916, -65.197, 123.895, -0.265, 52.003, -90.179, -98.001]
  MoveL 1780 to (-206.48, 49.48, -13.47) mm, rotated rx 180 ry 0 rz 74.1 deg; joints [-1.916, -65.183, 123.894, -0.266, 52.003, -90.178, -98.014]
  MoveL 1781 to (-206.43, 49.24, -13.48) mm, rotated rx 180 ry 0 rz 74.1 deg; joints [-1.916, -65.168, 123.892, -0.266, 52.003, -90.178, -98.027]
  MoveL 1782 to (-206.37, 49.02, -13.48) mm, rotated rx 180 ry 0 rz 74.1 deg; joints [-1.916, -65.153, 123.889, -0.266, 52.003, -90.178, -98.039]
  MoveL 1783 to (-206.28, 48.8, -13.48) mm, rotated rx 180 ry 0 rz 74.1 deg; joints [-1.916, -65.137, 123.884, -0.266, 52.003, -90.178, -98.05]
  MoveL 1784 to (-206.18, 48.57, -13.48) mm, rotated rx -180 ry 0 rz 74.1 deg; joints [-1.916, -65.12, 123.878, -0.266, 52.003, -90.178, -98.061]
  MoveL 1785 to (-206.06, 48.35, -13.48) mm, rotated rx 180 ry 0 rz 74.1 deg; joints [-1.916, -65.102, 123.871, -0.266, 52.003, -90.178, -98.072]
  MoveL 1786 to (-205.98, 48.22, -13.48) mm, rotated rx 180 ry 0 rz 74.1 deg; joints [-1.916, -65.091, 123.865, -0.266, 52.003, -90.178, -98.077]
  MoveL 1787 to (-205.88, 48.09, -13.48) mm, rotated rx -180 ry 0 rz 74.1 deg; joints [-1.916, -65.08, 123.86, -0.266, 52.003, -90.178, -98.083]
  MoveL 1788 to (-205.78, 47.96, -13.48) mm, rotated rx -180 ry 0 rz 74.1 deg; joints [-1.916, -65.068, 123.853, -0.266, 52.003, -90.178, -98.088]
  MoveL 1789 to (-205.66, 47.83, -13.48) mm, rotated rx 180 ry 0 rz 74.1 deg; joints [-1.916, -65.055, 123.845, -0.266, 52.003, -90.178, -98.093]
  MoveL 1790 to (-205.51, 47.67, -13.48) mm, rotated rx -180 ry 0 rz 74.1 deg; joints [-1.916, -65.038, 123.834, -0.266, 52.003, -90.178, -98.099]
  MoveL 1791 to (-205.35, 47.54, -13.48) mm, rotated rx -180 ry 0 rz 74.1 deg; joints [-1.916, -65.023, 123.824, -0.266, 52.003, -90.178, -98.104]
  MoveL 1792 to (-205.19, 47.42, -13.48) mm, rotated rx -180 ry 0 rz 74.1 deg; joints [-1.916, -65.008, 123.813, -0.266, 52.003, -90.177, -98.108]
  MoveL 1793 to (-205.03, 47.31, -13.48) mm, rotated rx -180 ry 0 rz 74.1 deg; joints [-1.916, -64.994, 123.802, -0.266, 52.003, -90.177, -98.11]
  MoveL 1794 to (-204.81, 47.18, -13.48) mm, rotated rx 180 ry 0 rz 74.1 deg; joints [-1.916, -64.976, 123.786, -0.266, 52.003, -90.177, -98.113]
  MoveL 1795 to (-204.58, 47.08, -13.48) mm, rotated rx -180 ry 0 rz 74.1 deg; joints [-1.915, -64.959, 123.77, -0.266, 52.003, -90.177, -98.114]
  MoveL 1796 to (-204.36, 46.99, -13.48) mm, rotated rx -180 ry 0 rz 74.1 deg; joints [-1.915, -64.942, 123.754, -0.266, 52.003, -90.177, -98.115]
  MoveL 1797 to (-204.13, 46.92, -13.48) mm, rotated rx -180 ry 0 rz 74.1 deg; joints [-1.915, -64.927, 123.737, -0.266, 52.003, -90.177, -98.114]
  MoveL 1798 to (-203.89, 46.87, -13.48) mm, rotated rx -180 ry 0 rz 74.1 deg; joints [-1.915, -64.911, 123.72, -0.266, 52.003, -90.177, -98.112]
  MoveL 1799 to (-203.65, 46.84, -13.48) mm, rotated rx -180 ry 0 rz 74.1 deg; joints [-1.915, -64.897, 123.702, -0.266, 52.003, -90.177, -98.108]
  MoveL 1800 to (-203.41, 46.83, -13.48) mm, rotated rx 180 ry 0 rz 74.1 deg; joints [-1.915, -64.884, 123.684, -0.266, 52.003, -90.177, -98.104]
  MoveL 1801 to (-203.17, 46.82, -13.48) mm, rotated rx -180 ry 0 rz 74.1 deg; joints [-1.915, -64.871, 123.666, -0.266, 52.003, -90.177, -98.099]
  MoveL 1802 to (222.09, 46.83, -13.48) mm, rotated rx -180 ry 0 rz 74.1 deg; joints [-1.822, -47.494, 88.471, -0.115, 52.003, -90.225, -80.28]
  MoveL 1803 to (223.29, 46.83, -13.48) mm, rotated rx 180 ry 0 rz 74.1 deg; joints [-1.822, -47.462, 88.363, -0.114, 52.003, -90.225, -80.203]
  MoveL 1804 to (223.53, 46.84, -13.48) mm, rotated rx 180 ry 0 rz 74.1 deg; joints [-1.822, -47.457, 88.341, -0.114, 52.003, -90.225, -80.188]
  MoveL 1805 to (223.77, 46.87, -13.47) mm, rotated rx 180 ry 0 rz 74.1 deg; joints [-1.821, -47.452, 88.32, -0.114, 52.003, -90.225, -80.171]
  MoveL 1806 to (224.01, 46.92, -13.48) mm, rotated rx 180 ry 0 rz 74.1 deg; joints [-1.821, -47.449, 88.299, -0.114, 52.003, -90.225, -80.153]
  MoveL 1807 to (224.24, 46.99, -13.48) mm, rotated rx -180 ry 0 rz 74.1 deg; joints [-1.821, -47.447, 88.28, -0.114, 52.003, -90.225, -80.136]
  MoveL 1808 to (224.46, 47.08, -13.47) mm, rotated rx -180 ry 0 rz 74.1 deg; joints [-1.821, -47.447, 88.262, -0.114, 52.003, -90.225, -80.118]
  MoveL 1809 to (224.69, 47.18, -13.48) mm, rotated rx 180 ry 0 rz 74.1 deg; joints [-1.821, -47.448, 88.244, -0.113, 52.003, -90.225, -80.099]
  MoveL 1810 to (224.92, 47.31, -13.48) mm, rotated rx -180 ry 0 rz 74.1 deg; joints [-1.821, -47.45, 88.226, -0.113, 52.002, -90.226, -80.079]
  MoveL 1811 to (225.07, 47.42, -13.48) mm, rotated rx 180 ry 0 rz 74.1 deg; joints [-1.821, -47.453, 88.214, -0.113, 52.003, -90.226, -80.064]
  MoveL 1812 to (225.23, 47.54, -13.47) mm, rotated rx -180 ry 0 rz 74.1 deg; joints [-1.821, -47.456, 88.202, -0.113, 52.002, -90.226, -80.049]
  MoveL 1813 to (225.39, 47.67, -13.48) mm, rotated rx 180 ry 0 rz 74.1 deg; joints [-1.821, -47.461, 88.191, -0.113, 52.002, -90.226, -80.033]
  MoveL 1814 to (225.55, 47.83, -13.48) mm, rotated rx 180 ry 0 rz 74.1 deg; joints [-1.821, -47.466, 88.18, -0.113, 52.002, -90.226, -80.016]
  MoveL 1815 to (225.66, 47.96, -13.48) mm, rotated rx -180 ry 0 rz 74.1 deg; joints [-1.821, -47.472, 88.172, -0.113, 52.002, -90.226, -80.003]
  MoveL 1816 to (225.77, 48.09, -13.48) mm, rotated rx 180 ry 0 rz 74.1 deg; joints [-1.821, -47.477, 88.165, -0.113, 52.002, -90.226, -79.991]
  MoveL 1817 to (225.86, 48.22, -13.47) mm, rotated rx 180 ry 0 rz 74.1 deg; joints [-1.821, -47.483, 88.16, -0.113, 52.002, -90.226, -79.979]
  MoveL 1818 to (225.94, 48.35, -13.48) mm, rotated rx -180 ry 0 rz 74.1 deg; joints [-1.821, -47.489, 88.155, -0.113, 52.002, -90.226, -79.968]
  MoveL 1819 to (226.07, 48.57, -13.48) mm, rotated rx -180 ry 0 rz 74.1 deg; joints [-1.821, -47.5, 88.148, -0.112, 52.002, -90.226, -79.951]
  MoveL 1820 to (226.17, 48.8, -13.47) mm, rotated rx -180 ry 0 rz 74.1 deg; joints [-1.821, -47.511, 88.144, -0.112, 52.002, -90.226, -79.935]
  MoveL 1821 to (226.25, 49.02, -13.48) mm, rotated rx -180 ry 0 rz 74.1 deg; joints [-1.821, -47.523, 88.141, -0.112, 52.002, -90.226, -79.92]
  MoveL 1822 to (226.31, 49.24, -13.48) mm, rotated rx 180 ry 0 rz 74.1 deg; joints [-1.821, -47.536, 88.14, -0.112, 52.002, -90.226, -79.906]
  MoveL 1823 to (226.36, 49.48, -13.48) mm, rotated rx 180 ry 0 rz 74.1 deg; joints [-1.821, -47.55, 88.14, -0.112, 52.002, -90.226, -79.893]
  MoveL 1824 to (226.39, 49.73, -13.47) mm, rotated rx -180 ry 0 rz 74.1 deg; joints [-1.821, -47.565, 88.142, -0.112, 52.002, -90.226, -79.88]
  MoveL 1825 to (226.4, 50.21, -13.47) mm, rotated rx -180 ry 0 rz 74.1 deg; joints [-1.821, -47.595, 88.151, -0.112, 52.002, -90.227, -79.859]
  MoveL 1826 to (226.4, 428.01, -13.47) mm, rotated rx 180 ry 0 rz 74.1 deg; joints [-1.826, -65.041, 88.151, -0.077, 66.065, -90.274, -76.476]
  MoveL 1827 to (226.4, 428.22, -13.47) mm, rotated rx -180 ry 0 rz 74.1 deg; joints [-1.826, -65.051, 88.151, -0.077, 66.072, -90.274, -76.471]
  MoveL 1828 to (226.38, 428.44, -13.48) mm, rotated rx -180 ry 0 rz 74.1 deg; joints [-1.826, -65.061, 88.151, -0.077, 66.079, -90.274, -76.469]
  MoveL 1829 to (226.35, 428.65, -13.48) mm, rotated rx 180 ry 0 rz 74.1 deg; joints [-1.826, -65.071, 88.151, -0.077, 66.088, -90.274, -76.468]
  MoveL 1830 to (226.3, 428.87, -13.47) mm, rotated rx -180 ry 0 rz 74.1 deg; joints [-1.826, -65.08, 88.151, -0.077, 66.099, -90.274, -76.47]
  MoveL 1831 to (226.24, 429.08, -13.48) mm, rotated rx -180 ry 0 rz 74.1 deg; joints [-1.826, -65.089, 88.151, -0.077, 66.111, -90.274, -76.473]
  MoveL 1832 to (226.16, 429.3, -13.47) mm, rotated rx -180 ry 0 rz 74.1 deg; joints [-1.826, -65.097, 88.151, -0.077, 66.125, -90.274, -76.479]
  MoveL 1833 to (226.06, 429.51, -13.47) mm, rotated rx -180 ry 0 rz 74.1 deg; joints [-1.826, -65.105, 88.151, -0.077, 66.14, -90.274, -76.487]
  MoveL 1834 to (225.94, 429.73, -13.47) mm, rotated rx -180 ry 0 rz 74.1 deg; joints [-1.826, -65.112, 88.151, -0.077, 66.158, -90.274, -76.497]
  MoveL 1835 to (225.8, 429.94, -13.47) mm, rotated rx -180 ry 0 rz 74.1 deg; joints [-1.826, -65.118, 88.151, -0.077, 66.177, -90.274, -76.51]
  MoveL 1836 to (225.6, 430.19, -13.47) mm, rotated rx 180 ry 0 rz 74.1 deg; joints [-1.826, -65.125, 88.151, -0.077, 66.204, -90.274, -76.53]
  MoveL 1837 to (225.35, 430.44, -13.47) mm, rotated rx 180 ry 0 rz 74.1 deg; joints [-1.826, -65.13, 88.151, -0.077, 66.234, -90.274, -76.556]
  MoveL 1838 to (225.13, 430.62, -13.47) mm, rotated rx -180 ry 0 rz 74.1 deg; joints [-1.826, -65.132, 88.151, -0.078, 66.261, -90.274, -76.58]
  MoveL 1839 to (224.91, 430.77, -13.47) mm, rotated rx -180 ry 0 rz 74.1 deg; joints [-1.826, -65.133, 88.151, -0.078, 66.286, -90.274, -76.604]
  MoveL 1840 to (224.68, 430.9, -13.47) mm, rotated rx 180 ry 0 rz 74.1 deg; joints [-1.826, -65.133, 88.152, -0.078, 66.31, -90.274, -76.629]
  MoveL 1841 to (224.46, 431, -13.47) mm, rotated rx -180 ry 0 rz 74.1 deg; joints [-1.826, -65.133, 88.153, -0.078, 66.332, -90.274, -76.653]
  MoveL 1842 to (224.24, 431.09, -13.47) mm, rotated rx -180 ry 0 rz 74.1 deg; joints [-1.826, -65.133, 88.156, -0.078, 66.352, -90.274, -76.676]
  MoveL 1843 to (224.01, 431.15, -13.47) mm, rotated rx -180 ry 0 rz 74.1 deg; joints [-1.826, -65.133, 88.16, -0.078, 66.37, -90.274, -76.697]
  MoveL 1844 to (223.77, 431.21, -13.48) mm, rotated rx -180 ry 0 rz 74.1 deg; joints [-1.826, -65.133, 88.166, -0.078, 66.387, -90.274, -76.72]
  MoveL 1845 to (223.53, 431.24, -13.47) mm, rotated rx -180 ry 0 rz 74.1 deg; joints [-1.826, -65.133, 88.173, -0.078, 66.402, -90.274, -76.742]
  MoveL 1846 to (223.29, 431.25, -13.47) mm, rotated rx 180 ry 0 rz 74.1 deg; joints [-1.826, -65.133, 88.18, -0.079, 66.415, -90.274, -76.763]
  MoveL 1847 to (223.05, 431.25, -13.47) mm, rotated rx -180 ry 0 rz 74.1 deg; joints [-1.826, -65.133, 88.189, -0.079, 66.427, -90.274, -76.783]
  MoveL 1848 to (-164.9, 431.25, -13.47) mm, rotated rx -180 ry 0 rz 74.1 deg; joints [-1.834, -65.133, 93.563, -0.261, 101.063, -90.244, -116.793]
  Set speed (38.1 mm/s)
  MoveL 1849 to (-165.25, 432.42, -13.47) mm, rotated rx 180 ry 0 rz 74.1 deg; joints [-1.834, -65.194, 93.551, -0.261, 101.063, -90.244, -116.721]
  MoveL 1850 to (-164.27, 433.07, -13.47) mm, rotated rx 180 ry 0 rz 74.1 deg; joints [-1.834, -65.194, 93.517, -0.261, 100.982, -90.244, -116.606]
  Set speed (25.4 mm/s)
  MoveL 1851 to (-164.27, 433.07, -15.84) mm, rotated rx -180 ry 0 rz 74.1 deg; joints [-1.925, -65.193, 93.517, -0.319, 100.98, -90.325, -116.604]
  MoveL 1852 to (-164.27, 432.44, -16.47) mm, rotated rx -180 ry 0 rz 74.1 deg; joints [-1.949, -65.173, 93.536, -0.335, 100.98, -90.347, -116.644]
  Set speed (38.1 mm/s)
  MoveL 1853 to (-164.9, 431.8, -16.47) mm, rotated rx -180 ry 0 rz 74.1 deg; joints [-1.949, -65.173, 93.572, -0.335, 101.021, -90.347, -116.72]
  Set speed (76.2 mm/s)
  MoveL 1854 to (-194.97, 431.8, -16.47) mm, rotated rx -180 ry 0 rz 74.1 deg; joints [-1.95, -65.501, 93.572, -0.353, 104.12, -90.353, -119.492]
  MoveL 1855 to (-199.31, 431.8, -16.48) mm, rotated rx -180 ry 0 rz 74.1 deg; joints [-1.95, -65.556, 93.572, -0.356, 104.558, -90.354, -119.875]
  MoveL 1856 to (-199.79, 431.8, -16.47) mm, rotated rx -180 ry 0 rz 74.1 deg; joints [-1.95, -65.562, 93.572, -0.356, 104.607, -90.354, -119.917]
  MoveL 1857 to (-200.03, 431.77, -16.48) mm, rotated rx 180 ry 0 rz 74.1 deg; joints [-1.95, -65.564, 93.572, -0.356, 104.632, -90.354, -119.941]
  MoveL 1858 to (-200.27, 431.73, -16.48) mm, rotated rx -180 ry 0 rz 74.1 deg; joints [-1.95, -65.565, 93.572, -0.357, 104.659, -90.354, -119.967]
  MoveL 1859 to (-200.52, 431.67, -16.47) mm, rotated rx -180 ry 0 rz 74.1 deg; joints [-1.95, -65.565, 93.572, -0.357, 104.685, -90.354, -119.994]
  MoveL 1860 to (-204.13, 430.52, -16.47) mm, rotated rx 180 ry 0 rz 74.1 deg; joints [-1.95, -65.565, 93.592, -0.359, 105.078, -90.355, -120.406]
  MoveL 1861 to (-204.42, 430.43, -16.48) mm, rotated rx -180 ry 0 rz 74.1 deg; joints [-1.95, -65.565, 93.594, -0.36, 105.109, -90.355, -120.439]
  MoveL 1862 to (-204.57, 430.37, -16.47) mm, rotated rx 180 ry 0 rz 74.1 deg; joints [-1.95, -65.565, 93.595, -0.36, 105.125, -90.355, -120.456]
  MoveL 1863 to (-204.72, 430.31, -16.47) mm, rotated rx -180 ry 0 rz 74.1 deg; joints [-1.95, -65.565, 93.598, -0.36, 105.14, -90.355, -120.473]
  MoveL 1864 to (-204.86, 430.23, -16.47) mm, rotated rx -180 ry 0 rz 74.1 deg; joints [-1.95, -65.565, 93.6, -0.36, 105.154, -90.355, -120.49]
  MoveL 1865 to (-205.01, 430.15, -16.47) mm, rotated rx -180 ry 0 rz 74.1 deg; joints [-1.95, -65.565, 93.604, -0.36, 105.168, -90.355, -120.508]
  MoveL 1866 to (-205.16, 430.05, -16.47) mm, rotated rx 180 ry 0 rz 74.1 deg; joints [-1.95, -65.565, 93.608, -0.36, 105.181, -90.355, -120.525]
  MoveL 1867 to (-205.3, 429.94, -16.47) mm, rotated rx -180 ry 0 rz 74.1 deg; joints [-1.95, -65.569, 93.617, -0.36, 105.188, -90.355, -120.537]
  MoveL 1868 to (-205.53, 429.75, -16.47) mm, rotated rx -180 ry 0 rz 74.1 deg; joints [-1.95, -65.569, 93.626, -0.36, 105.207, -90.355, -120.565]
  MoveL 1869 to (-205.75, 429.52, -16.47) mm, rotated rx 180 ry 0 rz 74.1 deg; joints [-1.95, -65.569, 93.638, -0.361, 105.223, -90.355, -120.593]
  MoveL 1870 to (-205.92, 429.3, -16.47) mm, rotated rx -180 ry 0 rz 74.1 deg; joints [-1.95, -65.569, 93.65, -0.361, 105.234, -90.355, -120.616]
  MoveL 1871 to (-206.06, 429.09, -16.47) mm, rotated rx 180 ry 0 rz 74.1 deg; joints [-1.95, -65.569, 93.662, -0.361, 105.241, -90.355, -120.635]
  MoveL 1872 to (-206.14, 428.95, -16.47) mm, rotated rx -180 ry 0 rz 74.1 deg; joints [-1.95, -65.569, 93.669, -0.361, 105.244, -90.355, -120.646]
  MoveL 1873 to (-206.21, 428.82, -16.48) mm, rotated rx -180 ry 0 rz 74.1 deg; joints [-1.95, -65.569, 93.677, -0.361, 105.246, -90.355, -120.656]
  MoveL 1874 to (-206.27, 428.69, -16.47) mm, rotated rx -180 ry 0 rz 74.1 deg; joints [-1.95, -65.569, 93.685, -0.361, 105.247, -90.355, -120.665]
  MoveL 1875 to (-206.32, 428.55, -16.47) mm, rotated rx -180 ry 0 rz 74.1 deg; joints [-1.95, -65.569, 93.694, -0.361, 105.247, -90.355, -120.673]
  MoveL 1876 to (-206.37, 428.42, -16.47) mm, rotated rx -180 ry 0 rz 74.1 deg; joints [-1.95, -65.568, 93.701, -0.361, 105.247, -90.355, -120.681]
  MoveL 1877 to (-206.41, 428.28, -16.47) mm, rotated rx -180 ry 0 rz 74.1 deg; joints [-1.95, -65.568, 93.709, -0.361, 105.247, -90.355, -120.689]
  MoveL 1878 to (-206.47, 428.01, -16.47) mm, rotated rx 180 ry 0 rz 74.1 deg; joints [-1.95, -65.564, 93.722, -0.361, 105.247, -90.355, -120.706]
  MoveL 1879 to (-206.5, 427.77, -16.47) mm, rotated rx -180 ry 0 rz 74.1 deg; joints [-1.95, -65.56, 93.733, -0.361, 105.247, -90.355, -120.721]
  MoveL 1880 to (-206.52, 427.53, -16.47) mm, rotated rx 180 ry 0 rz 74.1 deg; joints [-1.95, -65.555, 93.742, -0.361, 105.247, -90.355, -120.735]
  MoveL 1881 to (-206.52, 427.04, -16.47) mm, rotated rx 180 ry 0 rz 74.1 deg; joints [-1.95, -65.542, 93.759, -0.362, 105.247, -90.354, -120.765]
  MoveL 1882 to (-206.52, 50.21, -16.48) mm, rotated rx -180 ry 0 rz 74.1 deg; joints [-1.999, -60.47, 112.178, -0.486, 105.247, -90.246, -144.256]
  MoveL 1883 to (-206.51, 49.73, -16.48) mm, rotated rx 180 ry 0 rz 74.1 deg; joints [-1.999, -60.469, 112.207, -0.486, 105.247, -90.246, -144.285]
  MoveL 1884 to (-206.48, 49.48, -16.48) mm, rotated rx 180 ry 0 rz 74.1 deg; joints [-2, -60.467, 112.22, -0.486, 105.247, -90.245, -144.301]
  MoveL 1885 to (-206.43, 49.24, -16.48) mm, rotated rx 180 ry 0 rz 74.1 deg; joints [-2, -60.464, 112.233, -0.486, 105.247, -90.245, -144.317]
  MoveL 1886 to (-206.37, 49.02, -16.48) mm, rotated rx -180 ry 0 rz 74.1 deg; joints [-2, -60.459, 112.243, -0.486, 105.247, -90.245, -144.332]
  MoveL 1887 to (-206.28, 48.8, -16.48) mm, rotated rx -180 ry 0 rz 74.1 deg; joints [-2, -60.454, 112.253, -0.486, 105.247, -90.245, -144.347]
  MoveL 1888 to (-206.18, 48.57, -16.48) mm, rotated rx 180 ry 0 rz 74.1 deg; joints [-2, -60.447, 112.261, -0.486, 105.247, -90.245, -144.363]
  MoveL 1889 to (-206.06, 48.35, -16.48) mm, rotated rx -180 ry 0 rz 74.1 deg; joints [-2, -60.438, 112.269, -0.486, 105.247, -90.245, -144.379]
  MoveL 1890 to (-205.98, 48.22, -16.48) mm, rotated rx -180 ry 0 rz 74.1 deg; joints [-2, -60.432, 112.273, -0.486, 105.247, -90.245, -144.389]
  MoveL 1891 to (-205.88, 48.09, -16.48) mm, rotated rx 180 ry 0 rz 74.1 deg; joints [-2, -60.425, 112.276, -0.486, 105.247, -90.245, -144.399]
  MoveL 1892 to (-205.78, 47.96, -16.48) mm, rotated rx 180 ry 0 rz 74.1 deg; joints [-2, -60.418, 112.279, -0.486, 105.247, -90.245, -144.41]
  MoveL 1893 to (-205.66, 47.83, -16.48) mm, rotated rx -180 ry 0 rz 74.1 deg; joints [-2, -60.41, 112.282, -0.486, 105.247, -90.245, -144.42]
  MoveL 1894 to (-205.51, 47.67, -16.48) mm, rotated rx -180 ry 0 rz 74.1 deg; joints [-2, -60.398, 112.284, -0.486, 105.247, -90.245, -144.434]
  MoveL 1895 to (-205.35, 47.54, -16.48) mm, rotated rx 180 ry 0 rz 74.1 deg; joints [-2, -60.387, 112.285, -0.486, 105.247, -90.244, -144.446]
  MoveL 1896 to (-205.19, 47.42, -16.48) mm, rotated rx 180 ry 0 rz 74.1 deg; joints [-2, -60.376, 112.284, -0.486, 105.247, -90.244, -144.457]
  MoveL 1897 to (-205.03, 47.31, -16.48) mm, rotated rx -180 ry 0 rz 74.1 deg; joints [-2, -60.364, 112.283, -0.486, 105.247, -90.244, -144.467]
  MoveL 1898 to (-204.81, 47.18, -16.47) mm, rotated rx -180 ry 0 rz 74.1 deg; joints [-2, -60.348, 112.28, -0.486, 105.247, -90.244, -144.48]
  MoveL 1899 to (-204.58, 47.08, -16.48) mm, rotated rx -180 ry 0 rz 74.1 deg; joints [-2, -60.332, 112.276, -0.486, 105.247, -90.244, -144.492]
  MoveL 1900 to (-204.36, 46.99, -16.48) mm, rotated rx 180 ry 0 rz 74.1 deg; joints [-2, -60.316, 112.27, -0.486, 105.247, -90.244, -144.502]
  MoveL 1901 to (-204.13, 46.92, -16.48) mm, rotated rx 180 ry 0 rz 74.1 deg; joints [-2, -60.3, 112.263, -0.486, 105.247, -90.244, -144.512]
  MoveL 1902 to (-203.89, 46.87, -16.48) mm, rotated rx 180 ry 0 rz 74.1 deg; joints [-2, -60.282, 112.255, -0.486, 105.247, -90.244, -144.521]
  MoveL 1903 to (-203.65, 46.84, -16.48) mm, rotated rx 180 ry 0 rz 74.1 deg; joints [-2, -60.265, 112.245, -0.486, 105.247, -90.244, -144.528]
  MoveL 1904 to (-203.41, 46.83, -16.48) mm, rotated rx 180 ry 0 rz 74.1 deg; joints [-2, -60.248, 112.235, -0.486, 105.247, -90.244, -144.535]
  MoveL 1905 to (-203.17, 46.83, -16.48) mm, rotated rx -180 ry 0 rz 74.1 deg; joints [-2, -60.23, 112.223, -0.486, 105.247, -90.244, -144.541]
  MoveL 1906 to (222.09, 46.82, -16.48) mm, rotated rx -180 ry 0 rz 74.1 deg; joints [-1.944, -30.937, 88.679, -0.441, 105.247, -90.168, -150.289]
  MoveL 1907 to (223.29, 46.83, -16.48) mm, rotated rx 180 ry 0 rz 74.1 deg; joints [-1.944, -30.856, 88.593, -0.44, 105.247, -90.168, -150.284]
  MoveL 1908 to (223.53, 46.84, -16.47) mm, rotated rx 180 ry 0 rz 74.1 deg; joints [-1.944, -30.839, 88.574, -0.44, 105.247, -90.168, -150.282]
  MoveL 1909 to (223.77, 46.87, -16.48) mm, rotated rx 180 ry 0 rz 74.1 deg; joints [-1.943, -30.823, 88.553, -0.44, 105.247, -90.168, -150.277]
  MoveL 1910 to (224.01, 46.92, -16.48) mm, rotated rx -180 ry 0 rz 74.1 deg; joints [-1.943, -30.807, 88.53, -0.44, 105.247, -90.168, -150.271]
  MoveL 1911 to (224.24, 46.99, -16.47) mm, rotated rx 180 ry 0 rz 74.1 deg; joints [-1.943, -30.791, 88.506, -0.44, 105.247, -90.168, -150.262]
  MoveL 1912 to (224.46, 47.08, -16.47) mm, rotated rx -180 ry 0 rz 74.1 deg; joints [-1.943, -30.776, 88.48, -0.44, 105.247, -90.168, -150.252]
  MoveL 1913 to (224.69, 47.18, -16.47) mm, rotated rx -180 ry 0 rz 74.1 deg; joints [-1.943, -30.761, 88.452, -0.44, 105.247, -90.168, -150.239]
  MoveL 1914 to (224.92, 47.31, -16.47) mm, rotated rx -180 ry 0 rz 74.1 deg; joints [-1.943, -30.745, 88.422, -0.44, 105.247, -90.168, -150.224]
  MoveL 1915 to (225.07, 47.42, -16.47) mm, rotated rx -180 ry 0 rz 74.1 deg; joints [-1.943, -30.735, 88.398, -0.44, 105.247, -90.168, -150.211]
  MoveL 1916 to (225.23, 47.54, -16.48) mm, rotated rx 180 ry 0 rz 74.1 deg; joints [-1.943, -30.724, 88.373, -0.44, 105.247, -90.168, -150.197]
  MoveL 1917 to (225.39, 47.67, -16.47) mm, rotated rx 180 ry 0 rz 74.1 deg; joints [-1.943, -30.713, 88.346, -0.44, 105.247, -90.168, -150.181]
  MoveL 1918 to (225.55, 47.83, -16.47) mm, rotated rx -180 ry 0 rz 74.1 deg; joints [-1.943, -30.702, 88.317, -0.44, 105.247, -90.168, -150.163]
  MoveL 1919 to (225.66, 47.96, -16.47) mm, rotated rx -180 ry 0 rz 74.1 deg; joints [-1.943, -30.694, 88.294, -0.44, 105.247, -90.168, -150.148]
  MoveL 1920 to (225.77, 48.09, -16.47) mm, rotated rx 180 ry 0 rz 74.1 deg; joints [-1.943, -30.687, 88.272, -0.44, 105.247, -90.168, -150.133]
  MoveL 1921 to (225.86, 48.22, -16.47) mm, rotated rx -180 ry 0 rz 74.1 deg; joints [-1.943, -30.68, 88.251, -0.439, 105.247, -90.168, -150.118]
  MoveL 1922 to (225.94, 48.35, -16.47) mm, rotated rx -180 ry 0 rz 74.1 deg; joints [-1.943, -30.675, 88.23, -0.439, 105.247, -90.168, -150.103]
  MoveL 1923 to (226.07, 48.57, -16.47) mm, rotated rx -180 ry 0 rz 74.1 deg; joints [-1.943, -30.666, 88.196, -0.439, 105.247, -90.169, -150.077]
  MoveL 1924 to (226.17, 48.8, -16.48) mm, rotated rx -180 ry 0 rz 74.1 deg; joints [-1.943, -30.659, 88.163, -0.439, 105.247, -90.169, -150.052]
  MoveL 1925 to (226.25, 49.02, -16.47) mm, rotated rx 180 ry 0 rz 74.1 deg; joints [-1.942, -30.653, 88.132, -0.439, 105.247, -90.169, -150.027]
  MoveL 1926 to (226.31, 49.24, -16.47) mm, rotated rx -180 ry 0 rz 74.1 deg; joints [-1.942, -30.649, 88.102, -0.439, 105.247, -90.169, -150.001]
  MoveL 1927 to (226.36, 49.48, -16.48) mm, rotated rx 180 ry 0 rz 74.1 deg; joints [-1.942, -30.645, 88.072, -0.439, 105.247, -90.169, -149.974]
  MoveL 1928 to (226.39, 49.73, -16.48) mm, rotated rx -180 ry 0 rz 74.1 deg; joints [-1.942, -30.643, 88.042, -0.439, 105.247, -90.169, -149.947]
  MoveL 1929 to (226.4, 50.21, -16.47) mm, rotated rx -180 ry 0 rz 74.1 deg; joints [-1.942, -30.641, 87.987, -0.438, 105.247, -90.17, -149.893]
  MoveL 1930 to (226.4, 428.49, -16.47) mm, rotated rx 180 ry 0 rz 74.1 deg; joints [-1.877, -38.719, 59.244, -0.278, 105.247, -90.317, -113.073]
  MoveL 1931 to (226.4, 428.74, -16.47) mm, rotated rx -180 ry 0 rz 74.1 deg; joints [-1.877, -38.728, 59.235, -0.278, 105.247, -90.317, -113.054]
  MoveL 1932 to (226.38, 428.98, -16.47) mm, rotated rx -180 ry 0 rz 74.1 deg; joints [-1.876, -38.739, 59.227, -0.277, 105.247, -90.317, -113.036]
  MoveL 1933 to (226.35, 429.22, -16.47) mm, rotated rx 180 ry 0 rz 74.1 deg; joints [-1.876, -38.75, 59.222, -0.277, 105.247, -90.317, -113.019]
  MoveL 1934 to (226.29, 429.46, -16.47) mm, rotated rx -180 ry 0 rz 74.1 deg; joints [-1.876, -38.763, 59.218, -0.277, 105.247, -90.317, -113.003]
  MoveL 1935 to (226.22, 429.7, -16.47) mm, rotated rx 180 ry 0 rz 74.1 deg; joints [-1.876, -38.777, 59.217, -0.277, 105.247, -90.317, -112.988]
  MoveL 1936 to (226.12, 429.94, -16.48) mm, rotated rx -180 ry 0 rz 74.1 deg; joints [-1.876, -38.791, 59.217, -0.277, 105.248, -90.317, -112.975]
  MoveL 1937 to (226.04, 430.11, -16.47) mm, rotated rx -180 ry 0 rz 74.1 deg; joints [-1.877, -38.8, 59.217, -0.277, 105.251, -90.317, -112.969]
  MoveL 1938 to (225.94, 430.28, -16.47) mm, rotated rx -180 ry 0 rz 74.1 deg; joints [-1.877, -38.808, 59.217, -0.277, 105.256, -90.317, -112.965]
  MoveL 1939 to (225.86, 430.4, -16.48) mm, rotated rx 180 ry 0 rz 74.1 deg; joints [-1.877, -38.814, 59.217, -0.277, 105.261, -90.317, -112.964]
  MoveL 1940 to (225.77, 430.53, -16.47) mm, rotated rx -180 ry 0 rz 74.1 deg; joints [-1.877, -38.82, 59.217, -0.277, 105.267, -90.317, -112.965]
  MoveL 1941 to (225.67, 430.65, -16.47) mm, rotated rx -180 ry 0 rz 74.1 deg; joints [-1.877, -38.825, 59.217, -0.277, 105.274, -90.317, -112.967]
  MoveL 1942 to (225.57, 430.78, -16.48) mm, rotated rx -180 ry 0 rz 74.1 deg; joints [-1.877, -38.83, 59.217, -0.277, 105.283, -90.317, -112.972]
  MoveL 1943 to (225.42, 430.93, -16.47) mm, rotated rx 180 ry 0 rz 74.1 deg; joints [-1.877, -38.834, 59.217, -0.277, 105.297, -90.317, -112.98]
  MoveL 1944 to (225.27, 431.06, -16.48) mm, rotated rx -180 ry 0 rz 74.1 deg; joints [-1.877, -38.838, 59.217, -0.277, 105.311, -90.317, -112.991]
  MoveL 1945 to (225.12, 431.17, -16.47) mm, rotated rx 180 ry 0 rz 74.1 deg; joints [-1.877, -38.84, 59.217, -0.277, 105.326, -90.317, -113.004]
  MoveL 1946 to (224.98, 431.28, -16.47) mm, rotated rx -180 ry 0 rz 74.1 deg; joints [-1.877, -38.841, 59.217, -0.278, 105.342, -90.317, -113.019]
  MoveL 1947 to (224.74, 431.42, -16.47) mm, rotated rx -180 ry 0 rz 74.1 deg; joints [-1.877, -38.841, 59.218, -0.278, 105.369, -90.318, -113.046]
  MoveL 1948 to (224.5, 431.54, -16.47) mm, rotated rx 180 ry 0 rz 74.1 deg; joints [-1.877, -38.841, 59.22, -0.278, 105.394, -90.318, -113.074]
  MoveL 1949 to (224.25, 431.63, -16.47) mm, rotated rx 180 ry 0 rz 74.1 deg; joints [-1.877, -38.841, 59.224, -0.278, 105.418, -90.318, -113.102]
  MoveL 1950 to (224.01, 431.7, -16.47) mm, rotated rx -180 ry 0 rz 74.1 deg; joints [-1.877, -38.841, 59.23, -0.278, 105.441, -90.318, -113.13]
  MoveL 1951 to (223.77, 431.76, -16.48) mm, rotated rx -180 ry 0 rz 74.1 deg; joints [-1.877, -38.841, 59.237, -0.278, 105.463, -90.318, -113.159]
  MoveL 1952 to (223.53, 431.79, -16.47) mm, rotated rx -180 ry 0 rz 74.1 deg; joints [-1.877, -38.841, 59.246, -0.279, 105.484, -90.318, -113.189]
  MoveL 1953 to (223.29, 431.8, -16.47) mm, rotated rx -180 ry 0 rz 74.1 deg; joints [-1.877, -38.841, 59.256, -0.279, 105.504, -90.318, -113.219]
  MoveL 1954 to (223.05, 431.8, -16.47) mm, rotated rx -180 ry 0 rz 74.1 deg; joints [-1.877, -38.841, 59.267, -0.279, 105.523, -90.318, -113.249]
  MoveL 1955 to (-164.9, 431.8, -16.47) mm, rotated rx 180 ry 0 rz 74.1 deg; joints [-1.916, -54.896, 81.957, -0.421, 119, -90.362, -133.361]
  MoveL 1956 to (-194.97, 431.99, -17.52) mm, rotated rx 180 ry 0 rz 74.1 deg; joints [-1.958, -56.983, 83.816, -0.461, 119, -90.406, -133.134]
  MoveL 1957 to (-195.47, 431.99, -17.52) mm, rotated rx -180 ry 0 rz 74.1 deg; joints [-1.958, -57.017, 83.846, -0.461, 119, -90.407, -133.13]
  MoveL 1958 to (-198.35, 431.99, -17.52) mm, rotated rx -180 ry 0 rz 74.1 deg; joints [-1.959, -57.218, 84.023, -0.461, 119, -90.407, -133.106]
  MoveL 1959 to (-199.1, 431.99, -17.52) mm, rotated rx -180 ry 0 rz 74.1 deg; joints [-1.959, -57.27, 84.069, -0.461, 119, -90.407, -133.1]
  MoveL 1960 to (-199.28, 431.98, -17.52) mm, rotated rx -180 ry 0 rz 74.1 deg; joints [-1.959, -57.283, 84.081, -0.461, 119, -90.408, -133.1]
  MoveL 1961 to (-199.47, 431.96, -17.52) mm, rotated rx 180 ry 0 rz 74.1 deg; joints [-1.959, -57.296, 84.094, -0.461, 119, -90.408, -133.1]
  MoveL 1962 to (-199.66, 431.92, -17.52) mm, rotated rx -180 ry 0 rz 74.1 deg; joints [-1.959, -57.308, 84.107, -0.462, 119, -90.408, -133.1]
  MoveL 1963 to (-199.85, 431.88, -17.52) mm, rotated rx -180 ry 0 rz 74.1 deg; joints [-1.959, -57.321, 84.121, -0.462, 119, -90.408, -133.102]
  MoveL 1964 to (-200.27, 431.74, -17.52) mm, rotated rx -180 ry 0 rz 74.1 deg; joints [-1.959, -57.349, 84.154, -0.462, 119, -90.408, -133.107]
  MoveL 1965 to (-204.13, 430.52, -17.52) mm, rotated rx 180 ry 0 rz 74.1 deg; joints [-1.96, -57.601, 84.454, -0.463, 119, -90.408, -133.155]
  MoveL 1966 to (-204.42, 430.43, -17.52) mm, rotated rx 180 ry 0 rz 74.1 deg; joints [-1.96, -57.62, 84.477, -0.463, 119, -90.408, -133.159]
  MoveL 1967 to (-204.57, 430.37, -17.52) mm, rotated rx -180 ry 0 rz 74.1 deg; joints [-1.96, -57.629, 84.489, -0.463, 119, -90.408, -133.161]
  MoveL 1968 to (-204.72, 430.31, -17.52) mm, rotated rx -180 ry 0 rz 74.1 deg; joints [-1.96, -57.638, 84.501, -0.463, 119, -90.408, -133.164]
  MoveL 1969 to (-204.86, 430.23, -17.52) mm, rotated rx 180 ry 0 rz 74.1 deg; joints [-1.96, -57.648, 84.514, -0.463, 119, -90.408, -133.168]
  MoveL 1970 to (-205.01, 430.15, -17.52) mm, rotated rx -180 ry 0 rz 74.1 deg; joints [-1.96, -57.657, 84.527, -0.463, 119, -90.408, -133.172]
  MoveL 1971 to (-205.16, 430.05, -17.52) mm, rotated rx -180 ry 0 rz 74.1 deg; joints [-1.961, -57.665, 84.541, -0.463, 119, -90.408, -133.177]
  MoveL 1972 to (-205.3, 429.94, -17.52) mm, rotated rx 180 ry 0 rz 74.1 deg; joints [-1.961, -57.674, 84.556, -0.463, 119, -90.408, -133.183]
  MoveL 1973 to (-205.53, 429.75, -17.52) mm, rotated rx -180 ry 0 rz 74.1 deg; joints [-1.961, -57.687, 84.579, -0.463, 119, -90.408, -133.194]
  MoveL 1974 to (-205.75, 429.52, -17.52) mm, rotated rx 180 ry 0 rz 74.1 deg; joints [-1.961, -57.699, 84.605, -0.463, 119, -90.408, -133.207]
  MoveL 1975 to (-205.92, 429.3, -17.52) mm, rotated rx -180 ry 0 rz 74.1 deg; joints [-1.961, -57.708, 84.627, -0.463, 119, -90.408, -133.22]
  MoveL 1976 to (-206.06, 429.09, -17.52) mm, rotated rx -180 ry 0 rz 74.1 deg; joints [-1.961, -57.715, 84.646, -0.463, 119, -90.408, -133.233]
  MoveL 1977 to (-206.14, 428.95, -17.52) mm, rotated rx -180 ry 0 rz 74.1 deg; joints [-1.961, -57.719, 84.658, -0.463, 119, -90.408, -133.241]
  MoveL 1978 to (-206.21, 428.82, -17.52) mm, rotated rx -180 ry 0 rz 74.1 deg; joints [-1.961, -57.722, 84.669, -0.464, 119, -90.408, -133.249]
  MoveL 1979 to (-206.27, 428.69, -17.52) mm, rotated rx 180 ry 0 rz 74.1 deg; joints [-1.961, -57.724, 84.68, -0.464, 119, -90.408, -133.258]
  MoveL 1980 to (-206.32, 428.55, -17.52) mm, rotated rx 180 ry 0 rz 74.1 deg; joints [-1.961, -57.726, 84.69, -0.464, 119, -90.408, -133.266]
  MoveL 1981 to (-206.37, 428.42, -17.52) mm, rotated rx -180 ry 0 rz 74.1 deg; joints [-1.961, -57.727, 84.7, -0.464, 119, -90.408, -133.275]
  MoveL 1982 to (-206.41, 428.28, -17.52) mm, rotated rx -180 ry 0 rz 74.1 deg; joints [-1.961, -57.728, 84.71, -0.464, 119, -90.408, -133.283]
  MoveL 1983 to (-206.47, 428.01, -17.52) mm, rotated rx -180 ry 0 rz 74.1 deg; joints [-1.961, -57.729, 84.728, -0.464, 119, -90.408, -133.3]
  MoveL 1984 to (-206.5, 427.77, -17.52) mm, rotated rx 180 ry 0 rz 74.1 deg; joints [-1.961, -57.728, 84.742, -0.464, 119, -90.408, -133.316]
  MoveL 1985 to (-206.52, 427.53, -17.52) mm, rotated rx -180 ry 0 rz 74.1 deg; joints [-1.961, -57.725, 84.756, -0.464, 119, -90.408, -133.332]
  MoveL 1986 to (-206.52, 427.04, -17.52) mm, rotated rx 180 ry 0 rz 74.1 deg; joints [-1.961, -57.719, 84.781, -0.464, 119, -90.408, -133.364]
  MoveL 1987 to (-206.52, 50.21, -17.52) mm, rotated rx -180 ry 0 rz 74.1 deg; joints [-2.029, -58.042, 108.913, -0.585, 119, -90.299, -157.172]
  MoveL 1988 to (-206.51, 49.73, -17.52) mm, rotated rx -180 ry 0 rz 74.1 deg; joints [-2.029, -58.049, 108.947, -0.586, 119, -90.299, -157.2]
  MoveL 1989 to (-206.48, 49.48, -17.52) mm, rotated rx 180 ry 0 rz 74.1 deg; joints [-2.029, -58.05, 108.963, -0.586, 119, -90.299, -157.214]
  MoveL 1990 to (-206.43, 49.24, -17.52) mm, rotated rx -180 ry 0 rz 74.1 deg; joints [-2.029, -58.051, 108.979, -0.586, 119, -90.299, -157.23]
  MoveL 1991 to (-206.37, 49.02, -17.52) mm, rotated rx -180 ry 0 rz 74.1 deg; joints [-2.029, -58.05, 108.993, -0.586, 119, -90.299, -157.245]
  MoveL 1992 to (-206.28, 48.8, -17.52) mm, rotated rx -180 ry 0 rz 74.1 deg; joints [-2.029, -58.048, 109.006, -0.586, 119, -90.299, -157.26]
  MoveL 1993 to (-206.18, 48.57, -17.52) mm, rotated rx -180 ry 0 rz 74.1 deg; joints [-2.029, -58.044, 109.019, -0.586, 119, -90.299, -157.276]
  MoveL 1994 to (-206.06, 48.35, -17.52) mm, rotated rx -180 ry 0 rz 74.1 deg; joints [-2.029, -58.039, 109.031, -0.586, 119, -90.299, -157.293]
  MoveL 1995 to (-205.98, 48.22, -17.53) mm, rotated rx -180 ry 0 rz 74.1 deg; joints [-2.029, -58.035, 109.037, -0.586, 119, -90.299, -157.303]
  MoveL 1996 to (-205.88, 48.09, -17.52) mm, rotated rx -180 ry 0 rz 74.1 deg; joints [-2.029, -58.031, 109.043, -0.586, 119, -90.298, -157.314]
  MoveL 1997 to (-205.78, 47.96, -17.52) mm, rotated rx -180 ry 0 rz 74.1 deg; joints [-2.029, -58.026, 109.049, -0.586, 119, -90.298, -157.325]
  MoveL 1998 to (-205.66, 47.83, -17.52) mm, rotated rx 180 ry 0 rz 74.1 deg; joints [-2.029, -58.02, 109.055, -0.586, 119, -90.298, -157.336]
  MoveL 1999 to (-205.51, 47.67, -17.52) mm, rotated rx 180 ry 0 rz 74.1 deg; joints [-2.029, -58.011, 109.061, -0.586, 119, -90.298, -157.351]
  MoveL 2000 to (-205.35, 47.54, -17.52) mm, rotated rx 180 ry 0 rz 74.1 deg; joints [-2.03, -58.002, 109.065, -0.586, 119, -90.298, -157.364]
  MoveL 2001 to (-205.19, 47.42, -17.52) mm, rotated rx 180 ry 0 rz 74.1 deg; joints [-2.03, -57.993, 109.069, -0.586, 119, -90.298, -157.377]
  MoveL 2002 to (-205.03, 47.31, -17.52) mm, rotated rx -180 ry 0 rz 74.1 deg; joints [-2.03, -57.984, 109.071, -0.586, 119, -90.298, -157.388]
  MoveL 2003 to (-204.81, 47.18, -17.52) mm, rotated rx -180 ry 0 rz 74.1 deg; joints [-2.03, -57.97, 109.072, -0.586, 119, -90.298, -157.403]
  MoveL 2004 to (-204.58, 47.08, -17.52) mm, rotated rx 180 ry 0 rz 74.1 deg; joints [-2.03, -57.956, 109.072, -0.586, 119, -90.298, -157.417]
  MoveL 2005 to (-204.36, 46.99, -17.52) mm, rotated rx -180 ry 0 rz 74.1 deg; joints [-2.03, -57.942, 109.071, -0.586, 119, -90.297, -157.43]
  MoveL 2006 to (-204.13, 46.92, -17.52) mm, rotated rx -180 ry 0 rz 74.1 deg; joints [-2.03, -57.927, 109.068, -0.586, 119, -90.297, -157.442]
  MoveL 2007 to (-203.89, 46.87, -17.52) mm, rotated rx -180 ry 0 rz 74.1 deg; joints [-2.029, -57.911, 109.063, -0.586, 119, -90.297, -157.453]
  MoveL 2008 to (-203.65, 46.84, -17.52) mm, rotated rx -180 ry 0 rz 74.1 deg; joints [-2.029, -57.895, 109.058, -0.586, 119, -90.297, -157.464]
  MoveL 2009 to (-203.41, 46.83, -17.52) mm, rotated rx 180 ry 0 rz 74.1 deg; joints [-2.029, -57.878, 109.05, -0.586, 119, -90.297, -157.473]
  MoveL 2010 to (-203.17, 46.82, -17.53) mm, rotated rx 180 ry 0 rz 74.1 deg; joints [-2.029, -57.862, 109.042, -0.586, 119, -90.297, -157.482]
  MoveL 2011 to (222.09, 46.83, -17.52) mm, rotated rx 180 ry 0 rz 54.1 deg; joints [-2.009, -65.582, 101.118, 0.515, 22.306, -90.928, -25.14]
  MoveL 2012 to (223.29, 46.83, -17.52) mm, rotated rx -180 ry 0 rz 74.1 deg; joints [-2.012, -29.96, 96.373, -0.55, 119, -90.146, -172.713]
  MoveL 2013 to (223.53, 46.84, -17.52) mm, rotated rx -180 ry 0 rz 74.1 deg; joints [-2.012, -29.945, 96.365, -0.549, 119, -90.146, -172.72]
  MoveL 2014 to (223.77, 46.87, -17.52) mm, rotated rx -180 ry 0 rz 74.1 deg; joints [-2.012, -29.929, 96.355, -0.549, 119, -90.146, -172.726]
  MoveL 2015 to (224.01, 46.92, -17.53) mm, rotated rx 180 ry 0 rz 74.1 deg; joints [-2.012, -29.913, 96.342, -0.549, 119, -90.146, -172.73]
  MoveL 2016 to (224.24, 46.99, -17.52) mm, rotated rx -180 ry 0 rz 74.1 deg; joints [-2.012, -29.897, 96.328, -0.549, 119, -90.146, -172.731]
  MoveL 2017 to (224.46, 47.08, -17.52) mm, rotated rx -180 ry 0 rz 74.1 deg; joints [-2.012, -29.881, 96.311, -0.549, 119, -90.146, -172.731]
  MoveL 2018 to (224.69, 47.18, -17.52) mm, rotated rx -180 ry 0 rz 74.1 deg; joints [-2.012, -29.864, 96.291, -0.549, 119, -90.146, -172.728]
  MoveL 2019 to (224.92, 47.31, -17.52) mm, rotated rx -180 ry 0 rz 74.1 deg; joints [-2.012, -29.847, 96.269, -0.549, 119, -90.146, -172.723]
  MoveL 2020 to (225.07, 47.42, -17.53) mm, rotated rx -180 ry 0 rz 74.1 deg; joints [-2.012, -29.834, 96.251, -0.549, 119, -90.146, -172.717]
  MoveL 2021 to (225.23, 47.54, -17.52) mm, rotated rx 180 ry 0 rz 74.1 deg; joints [-2.012, -29.821, 96.23, -0.549, 119, -90.146, -172.71]
  MoveL 2022 to (225.39, 47.67, -17.52) mm, rotated rx 180 ry 0 rz 74.1 deg; joints [-2.012, -29.807, 96.208, -0.549, 119, -90.146, -172.701]
  MoveL 2023 to (225.55, 47.83, -17.53) mm, rotated rx -180 ry 0 rz 74.1 deg; joints [-2.012, -29.793, 96.183, -0.549, 119, -90.146, -172.69]
  MoveL 2024 to (225.66, 47.96, -17.52) mm, rotated rx -180 ry 0 rz 74.1 deg; joints [-2.012, -29.783, 96.163, -0.549, 119, -90.146, -172.681]
  MoveL 2025 to (225.77, 48.09, -17.52) mm, rotated rx -180 ry 0 rz 74.1 deg; joints [-2.011, -29.773, 96.142, -0.549, 119, -90.146, -172.67]
  MoveL 2026 to (225.86, 48.22, -17.52) mm, rotated rx 180 ry 0 rz 74.1 deg; joints [-2.011, -29.763, 96.123, -0.549, 119, -90.146, -172.66]
  MoveL 2027 to (225.94, 48.35, -17.52) mm, rotated rx 180 ry 0 rz 74.1 deg; joints [-2.011, -29.755, 96.103, -0.549, 119, -90.146, -172.649]
  MoveL 2028 to (226.07, 48.57, -17.52) mm, rotated rx -180 ry 0 rz 74.1 deg; joints [-2.011, -29.741, 96.07, -0.549, 119, -90.146, -172.629]
  MoveL 2029 to (226.17, 48.8, -17.52) mm, rotated rx 180 ry 0 rz 74.1 deg; joints [-2.011, -29.729, 96.037, -0.549, 119, -90.146, -172.609]
  MoveL 2030 to (226.25, 49.02, -17.52) mm, rotated rx -180 ry 0 rz 74.1 deg; joints [-2.011, -29.718, 96.005, -0.549, 119, -90.146, -172.588]
  MoveL 2031 to (226.31, 49.24, -17.52) mm, rotated rx 180 ry 0 rz 74.1 deg; joints [-2.011, -29.708, 95.973, -0.549, 119, -90.147, -172.566]
  MoveL 2032 to (226.36, 49.48, -17.52) mm, rotated rx -180 ry 0 rz 74.1 deg; joints [-2.011, -29.698, 95.939, -0.549, 119, -90.147, -172.541]
  MoveL 2033 to (226.39, 49.73, -17.52) mm, rotated rx -180 ry 0 rz 74.1 deg; joints [-2.011, -29.69, 95.905, -0.549, 119, -90.147, -172.516]
  MoveL 2034 to (226.4, 50.21, -17.52) mm, rotated rx 180 ry 0 rz 74.1 deg; joints [-2.01, -29.676, 95.839, -0.548, 119, -90.147, -172.464]
  MoveL 2035 to (226.4, 428.01, -17.52) mm, rotated rx -180 ry 0 rz 54.1 deg; joints [-2.034, -76.93, 101.191, -0.002, 57.613, -90.517, -49.174]
  MoveL 2036 to (226.4, 428.98, -17.52) mm, rotated rx 180 ry 0 rz 74.1 deg; joints [-1.899, -29.701, 50.703, -0.379, 118.218, -90.369, -126.521]
  MoveL 2037 to (226.38, 429.22, -17.53) mm, rotated rx -180 ry 0 rz 74.1 deg; joints [-1.899, -29.708, 50.686, -0.379, 118.218, -90.369, -126.497]
  MoveL 2038 to (226.34, 429.46, -17.52) mm, rotated rx -180 ry 0 rz 74.1 deg; joints [-1.899, -29.717, 50.672, -0.379, 118.218, -90.369, -126.475]
  MoveL 2039 to (226.28, 429.7, -17.52) mm, rotated rx -180 ry 0 rz 74.1 deg; joints [-1.899, -29.727, 50.661, -0.379, 118.218, -90.369, -126.453]
  MoveL 2040 to (226.2, 429.94, -17.52) mm, rotated rx -180 ry 0 rz 74.1 deg; joints [-1.899, -29.738, 50.651, -0.379, 118.218, -90.369, -126.433]
  MoveL 2041 to (226.15, 430.07, -17.52) mm, rotated rx 180 ry 0 rz 74.1 deg; joints [-1.899, -29.745, 50.647, -0.379, 118.218, -90.369, -126.422]
  MoveL 2042 to (226.09, 430.21, -17.52) mm, rotated rx 180 ry 0 rz 74.1 deg; joints [-1.899, -29.752, 50.644, -0.379, 118.218, -90.369, -126.412]
  MoveL 2043 to (226.02, 430.34, -17.52) mm, rotated rx -180 ry 0 rz 74.1 deg; joints [-1.899, -29.759, 50.642, -0.379, 118.218, -90.369, -126.402]
  MoveL 2044 to (225.94, 430.47, -17.52) mm, rotated rx -180 ry 0 rz 74.1 deg; joints [-1.899, -29.768, 50.641, -0.379, 118.218, -90.369, -126.392]
  MoveL 2045 to (225.78, 430.71, -17.52) mm, rotated rx -180 ry 0 rz 74.1 deg; joints [-1.899, -29.784, 50.641, -0.379, 118.218, -90.369, -126.376]
  MoveL 2046 to (225.58, 430.96, -17.52) mm, rotated rx -180 ry 0 rz 74.1 deg; joints [-1.899, -29.798, 50.641, -0.379, 118.226, -90.369, -126.369]
  MoveL 2047 to (225.44, 431.1, -17.52) mm, rotated rx -180 ry 0 rz 74.1 deg; joints [-1.899, -29.805, 50.641, -0.379, 118.234, -90.369, -126.371]
  MoveL 2048 to (225.3, 431.23, -17.52) mm, rotated rx 180 ry 0 rz 74.1 deg; joints [-1.899, -29.809, 50.641, -0.379, 118.244, -90.37, -126.377]
  MoveL 2049 to (225.16, 431.34, -17.52) mm, rotated rx -180 ry 0 rz 74.1 deg; joints [-1.899, -29.813, 50.64, -0.379, 118.257, -90.37, -126.386]
  MoveL 2050 to (225.02, 431.44, -17.52) mm, rotated rx -180 ry 0 rz 74.1 deg; joints [-1.899, -29.814, 50.64, -0.379, 118.27, -90.37, -126.397]
  MoveL 2051 to (224.78, 431.59, -17.52) mm, rotated rx -180 ry 0 rz 74.1 deg; joints [-1.899, -29.815, 50.64, -0.379, 118.296, -90.37, -126.423]
  MoveL 2052 to (224.55, 431.71, -17.52) mm, rotated rx -180 ry 0 rz 74.1 deg; joints [-1.899, -29.815, 50.643, -0.379, 118.321, -90.37, -126.45]
  MoveL 2053 to (224.32, 431.8, -17.52) mm, rotated rx -180 ry 0 rz 74.1 deg; joints [-1.899, -29.815, 50.647, -0.38, 118.346, -90.37, -126.479]
  MoveL 2054 to (224.09, 431.88, -17.52) mm, rotated rx 180 ry 0 rz 74.1 deg; joints [-1.899, -29.817, 50.655, -0.38, 118.367, -90.37, -126.506]
  MoveL 2055 to (224.01, 431.9, -17.52) mm, rotated rx 180 ry 0 rz 74.1 deg; joints [-1.899, -29.817, 50.657, -0.38, 118.374, -90.37, -126.516]
  MoveL 2056 to (223.77, 431.95, -17.52) mm, rotated rx -180 ry 0 rz 74.1 deg; joints [-1.899, -29.817, 50.667, -0.38, 118.398, -90.37, -126.549]
  MoveL 2057 to (223.53, 431.98, -17.52) mm, rotated rx -180 ry 0 rz 74.1 deg; joints [-1.899, -29.817, 50.678, -0.38, 118.421, -90.37, -126.583]
  MoveL 2058 to (223.29, 431.99, -17.52) mm, rotated rx 180 ry 0 rz 74.1 deg; joints [-1.899, -29.817, 50.691, -0.38, 118.443, -90.37, -126.618]
  MoveL 2059 to (223.05, 431.99, -17.52) mm, rotated rx -180 ry 0 rz 74.1 deg; joints [-1.899, -29.817, 50.705, -0.381, 118.465, -90.37, -126.654]
  MoveL 2060 to (-164.9, 431.99, -17.52) mm, rotated rx -180 ry 0 rz 74.1 deg; joints [-1.953, -54.899, 81.945, -0.456, 119, -90.4, -133.348]
  MoveL 2061 to (-194.97, 431.99, -17.52) mm, rotated rx 180 ry 0 rz 74.1 deg; joints [-1.958, -56.983, 83.815, -0.461, 119, -90.406, -133.134]
  MoveL 2062 to (-195.47, 431.99, -17.52) mm, rotated rx -180 ry 0 rz 74.1 deg; joints [-1.958, -57.017, 83.846, -0.461, 119, -90.407, -133.13]
  Set speed (38.1 mm/s)
  MoveL 2063 to (-196.09, 432.77, -17.52) mm, rotated rx -180 ry 0 rz 74.1 deg; joints [-1.959, -57.072, 83.844, -0.461, 119, -90.407, -133.073]
  MoveL 2064 to (-195.65, 434.72, -17.52) mm, rotated rx -180 ry 0 rz 74.1 deg; joints [-1.958, -57.072, 83.717, -0.46, 118.996, -90.407, -132.943]
  MoveL 2065 to (-195.51, 435.34, -16.89) mm, rotated rx -180 ry 0 rz 74.1 deg; joints [-1.936, -57.072, 83.677, -0.438, 118.996, -90.384, -132.902]
  Set speed (100.0 mm/s)
  MoveL 2066 to (-195.51, 435.34, 34.52) mm, rotated rx 180 ry 0 rz 74.1 deg; joints [-0.106, -57.072, 83.667, 1.286, 118.944, -88.515, -132.852]
  MoveL 2067 to (-195.51, 435.34, 34.52) mm, rotated rx 180 ry 0 rz 74.1 deg; joints [-0.106, -57.072, 83.667, 1.286, 118.944, -88.515, -132.852]

--- program sync move test (robot KUKA KR 30 HA) ---
  Smooth(10)
  Set Ref.: Frame 5
  Set Tool: rc90 spindle mm
  MoveJ (Target 1)
  MoveL (Target 2)
